LIN {X 0,Y 573.247,Z 310.075,A -85,B 0,C 180,E1 -2008.028,E2 -2008.028} C_VEL
LIN {X 0,Y 573.239,Z 310.078,A -85,B 0,C 180,E1 -2010.176,E2 -2010.176} C_VEL
LIN {X 0,Y 573.253,Z 310.082,A -85,B 0,C 180,E1 -2012.645,E2 -2012.645} C_VEL
LIN {X 0,Y 573.206,Z 310.08,A -85,B 0,C 180,E1 -2015.187,E2 -2015.187} C_VEL
LIN {X 0,Y 573.233,Z 310.076,A -85,B 0,C 180,E1 -2017.807,E2 -2017.807} C_VEL
LIN {X 0,Y 573.244,Z 310.084,A -85,B 0,C 180,E1 -2020.525,E2 -2020.525} C_VEL
LIN {X 0,Y 573.239,Z 310.074,A -85,B 0,C 180,E1 -2023.359,E2 -2023.359} C_VEL
LIN {X 0,Y 573.237,Z 310.083,A -85,B 0,C 180,E1 -2026.331,E2 -2026.331} C_VEL
LIN {X 0,Y 573.228,Z 310.084,A -85,B 0,C 180,E1 -2028.543,E2 -2028.543} C_VEL
LIN {X 0,Y 573.246,Z 310.073,A -85,B 0,C 180,E1 -2031.299,E2 -2031.299} C_VEL
LIN {X 0,Y 573.241,Z 310.079,A -85,B 0,C 180,E1 -2034.014,E2 -2034.014} C_VEL
LIN {X 0,Y 573.284,Z 310.076,A -85,B 0,C 180,E1 -2036.519,E2 -2036.519} C_VEL
LIN {X 0,Y 573.236,Z 310.075,A -85,B 0,C 180,E1 -2039.116,E2 -2039.116} C_VEL
LIN {X 0,Y 573.25,Z 310.078,A -85,B 0,C 180,E1 -2041.971,E2 -2041.971} C_VEL
LIN {X 0,Y 573.255,Z 310.077,A -85,B 0,C 180,E1 -2044.59,E2 -2044.59} C_VEL
LIN {X 0,Y 573.234,Z 310.077,A -85,B 0,C 180,E1 -2047.662,E2 -2047.662} C_VEL
LIN {X 0,Y 573.276,Z 310.072,A -85,B 0,C 180,E1 -2050.728,E2 -2050.728} C_VEL
LIN {X 0,Y 573.247,Z 310.076,A -85,B 0,C 180,E1 -2053.622,E2 -2053.622} C_VEL
LIN {X 0,Y 573.272,Z 310.075,A -85,B 0,C 180,E1 -2055.807,E2 -2055.807} C_VEL
LIN {X 0,Y 573.26,Z 310.073,A -85,B 0,C 180,E1 -2058.745,E2 -2058.745} C_VEL
LIN {X 0,Y 573.282,Z 310.071,A -85,B 0,C 180,E1 -2061.541,E2 -2061.541} C_VEL
LIN {X 0,Y 573.29,Z 310.073,A -85,B 0,C 180,E1 -2064.372,E2 -2064.372} C_VEL
LIN {X 0,Y 573.313,Z 310.073,A -85,B 0,C 180,E1 -2067.893,E2 -2067.893} C_VEL
LIN {X 0,Y 573.33,Z 310.064,A -85,B 0,C 180,E1 -2070.702,E2 -2070.702} C_VEL
LIN {X 0,Y 573.302,Z 310.067,A -85,B 0,C 180,E1 -2072.811,E2 -2072.811} C_VEL
LIN {X 0,Y 573.29,Z 310.073,A -85,B 0,C 180,E1 -2075.628,E2 -2075.628} C_VEL
LIN {X 0,Y 573.282,Z 310.071,A -85,B 0,C 180,E1 -2078.46,E2 -2078.46} C_VEL
LIN {X 0,Y 573.27,Z 310.072,A -85,B 0,C 180,E1 -2081.312,E2 -2081.312} C_VEL
LIN {X 0,Y 573.28,Z 310.071,A -85,B 0,C 180,E1 -2084.425,E2 -2084.425} C_VEL
LIN {X 0,Y 573.258,Z 310.073,A -85,B 0,C 180,E1 -2087.112,E2 -2087.112} C_VEL
LIN {X 0,Y 573.25,Z 310.079,A -85,B 0,C 180,E1 -2090.077,E2 -2090.077} C_VEL
LIN {X 0,Y 573.233,Z 310.076,A -85,B 0,C 180,E1 -2093.1,E2 -2093.1} C_VEL
LIN {X 0,Y 573.255,Z 310.077,A -85,B 0,C 180,E1 -2095.41,E2 -2095.41} C_VEL
LIN {X 0,Y 573.252,Z 310.078,A -85,B 0,C 180,E1 -2098.03,E2 -2098.03} C_VEL
LIN {X 0,Y 573.237,Z 310.075,A -85,B 0,C 180,E1 -2100.884,E2 -2100.884} C_VEL
LIN {X 0,Y 573.262,Z 310.079,A -85,B 0,C 180,E1 -2103.524,E2 -2103.524} C_VEL
LIN {X 0,Y 573.241,Z 310.078,A -85,B 0,C 180,E1 -2106.05,E2 -2106.05} C_VEL
LIN {X 0,Y 573.248,Z 310.073,A -85,B 0,C 180,E1 -2108.702,E2 -2108.702} C_VEL
LIN {X 0,Y 573.229,Z 310.085,A -85,B 0,C 180,E1 -2111.593,E2 -2111.593} C_VEL
LIN {X 0,Y 573.225,Z 310.077,A -85,B 0,C 180,E1 -2114.335,E2 -2114.335} C_VEL
LIN {X 0,Y 573.242,Z 310.081,A -85,B 0,C 180,E1 -2117.359,E2 -2117.359} C_VEL
LIN {X 0,Y 573.24,Z 310.075,A -85,B 0,C 180,E1 -2120.393,E2 -2120.393} C_VEL
LIN {X 0,Y 573.253,Z 310.076,A -85,B 0,C 180,E1 -2123.078,E2 -2123.078} C_VEL
LIN {X 0,Y 573.263,Z 310.078,A -85,B 0,C 180,E1 -2125.671,E2 -2125.671} C_VEL
LIN {X 0,Y 573.241,Z 310.075,A -85,B 0,C 180,E1 -2128.185,E2 -2128.185} C_VEL
LIN {X 0,Y 573.262,Z 310.072,A -85,B 0,C 180,E1 -2130.634,E2 -2130.634} C_VEL
LIN {X 0,Y 573.238,Z 310.083,A -85,B 0,C 180,E1 -2133.509,E2 -2133.509} C_VEL
LIN {X 0,Y 573.225,Z 310.077,A -85,B 0,C 180,E1 -2136.135,E2 -2136.135} C_VEL
LIN {X 0,Y 573.249,Z 310.075,A -85,B 0,C 180,E1 -2138.421,E2 -2138.421} C_VEL
LIN {X 0,Y 573.964,Z 312.69,A -85,B 0,C 180,E1 -2138.478,E2 -2138.478} C_VEL
LIN {X 0,Y 573.861,Z 400.24,A -85,B 0,C 180,E1 -2139.595,E2 -2139.595} C_VEL
LIN {X 0,Y 573.825,Z 411.853,A -85,B 0,C 180,E1 -2139.851,E2 -2139.851} C_VEL
LIN {X 0,Y 573.712,Z 424.112,A -85,B 0,C 180,E1 -2140.248,E2 -2140.248} C_VEL
LIN {X 0,Y 573.584,Z 437.638,A -85,B 0,C 180,E1 -2140.867,E2 -2140.867} C_VEL
LIN {X 0,Y 573.443,Z 448.401,A -85,B 0,C 180,E1 -2141.512,E2 -2141.512} C_VEL
LIN {X 0,Y 573.364,Z 457.219,A -85,B 0,C 180,E1 -2142.156,E2 -2142.156} C_VEL
LIN {X 0,Y 573.312,Z 465.622,A -85,B 0,C 180,E1 -2142.89,E2 -2142.89} C_VEL
LIN {X 0,Y 573.205,Z 472.699,A -85,B 0,C 180,E1 -2143.621,E2 -2143.621} C_VEL
LIN {X 0,Y 573.128,Z 480.104,A -85,B 0,C 180,E1 -2144.532,E2 -2144.532} C_VEL
LIN {X 0,Y 573.081,Z 486.335,A -85,B 0,C 180,E1 -2145.457,E2 -2145.457} C_VEL
LIN {X 0,Y 573.039,Z 492.198,A -85,B 0,C 180,E1 -2146.525,E2 -2146.525} C_VEL
LIN {X 0,Y 573.011,Z 496.871,A -85,B 0,C 180,E1 -2147.606,E2 -2147.606} C_VEL
LIN {X 0,Y 572.987,Z 500.957,A -85,B 0,C 180,E1 -2148.888,E2 -2148.888} C_VEL
LIN {X 0,Y 572.974,Z 503.485,A -85,B 0,C 180,E1 -2150.112,E2 -2150.112} C_VEL
LIN {X 0,Y 572.927,Z 504.386,A -85,B 0,C 180,E1 -2150.824,E2 -2150.824} C_VEL
LIN {X 0,Y 572.978,Z 504.962,A -85,B 0,C 180,E1 -2152.246,E2 -2152.246} C_VEL
LIN {X 0,Y 573.012,Z 504.176,A -85,B 0,C 180,E1 -2153.451,E2 -2153.451} C_VEL
LIN {X 0,Y 573,Z 502.806,A -85,B 0,C 180,E1 -2154.369,E2 -2154.369} C_VEL
LIN {X 0,Y 573.004,Z 500.334,A -85,B 0,C 180,E1 -2155.428,E2 -2155.428} C_VEL
LIN {X 0,Y 573.054,Z 496.866,A -85,B 0,C 180,E1 -2156.485,E2 -2156.485} C_VEL
LIN {X 0,Y 573.033,Z 492.323,A -85,B 0,C 180,E1 -2157.54,E2 -2157.54} C_VEL
LIN {X 0,Y 573.037,Z 486.574,A -85,B 0,C 180,E1 -2158.595,E2 -2158.595} C_VEL
LIN {X 0,Y 573.133,Z 480.729,A -85,B 0,C 180,E1 -2159.473,E2 -2159.473} C_VEL
LIN {X 0,Y 573.178,Z 473.733,A -85,B 0,C 180,E1 -2160.352,E2 -2160.352} C_VEL
LIN {X 0,Y 573.283,Z 465.315,A -85,B 0,C 180,E1 -2161.23,E2 -2161.23} C_VEL
LIN {X 0,Y 573.381,Z 456.163,A -85,B 0,C 180,E1 -2162.02,E2 -2162.02} C_VEL
LIN {X 0,Y 573.481,Z 444.879,A -85,B 0,C 180,E1 -2162.81,E2 -2162.81} C_VEL
LIN {X 0,Y 573.648,Z 433.661,A -85,B 0,C 180,E1 -2163.424,E2 -2163.424} C_VEL
LIN {X 0,Y 573.725,Z 422.252,A -85,B 0,C 180,E1 -2163.907,E2 -2163.907} C_VEL
LIN {X 0,Y 573.768,Z 411.124,A -85,B 0,C 180,E1 -2164.259,E2 -2164.259} C_VEL
LIN {X 0,Y 573.82,Z 399.944,A -85,B 0,C 180,E1 -2164.5,E2 -2164.5} C_VEL
LIN {X 0,Y 573.937,Z 312.624,A -85,B 0,C 180,E1 -2165.614,E2 -2165.614} C_VEL
LIN {X 0,Y 573.248,Z 310.076,A -85,B 0,C 180,E1 -2165.673,E2 -2165.673} C_VEL
LIN {X 0,Y 573.237,Z 310.083,A -85,B 0,C 180,E1 -2168.461,E2 -2168.461} C_VEL
LIN {X 0,Y 573.238,Z 310.076,A -85,B 0,C 180,E1 -2171.313,E2 -2171.313} C_VEL
LIN {X 0,Y 573.262,Z 310.081,A -85,B 0,C 180,E1 -2174.414,E2 -2174.414} C_VEL
LIN {X 0,Y 573.221,Z 310.079,A -85,B 0,C 180,E1 -2177.113,E2 -2177.113} C_VEL
LIN {X 0,Y 573.193,Z 310.086,A -85,B 0,C 180,E1 -2180.079,E2 -2180.079} C_VEL
LIN {X 0,Y 573.223,Z 310.077,A -85,B 0,C 180,E1 -2183.1,E2 -2183.1} C_VEL
LIN {X 0,Y 573.203,Z 310.08,A -85,B 0,C 180,E1 -2185.413,E2 -2185.413} C_VEL
LIN {X 0,Y 573.195,Z 310.087,A -85,B 0,C 180,E1 -2188.017,E2 -2188.017} C_VEL
LIN {X 0,Y 573.216,Z 310.078,A -85,B 0,C 180,E1 -2190.879,E2 -2190.879} C_VEL
LIN {X 0,Y 573.247,Z 310.075,A -85,B 0,C 180,E1 -2193.521,E2 -2193.521} C_VEL
LIN {X 0,Y 573.188,Z 310.09,A -85,B 0,C 180,E1 -2196.054,E2 -2196.054} C_VEL
LIN {X 0,Y 573.234,Z 310.075,A -85,B 0,C 180,E1 -2198.703,E2 -2198.703} C_VEL
LIN {X 0,Y 573.207,Z 310.081,A -85,B 0,C 180,E1 -2201.459,E2 -2201.459} C_VEL
LIN {X 0,Y 573.221,Z 310.08,A -85,B 0,C 180,E1 -2204.335,E2 -2204.335} C_VEL
LIN {X 0,Y 573.233,Z 310.079,A -85,B 0,C 180,E1 -2207.36,E2 -2207.36} C_VEL
LIN {X 0,Y 573.239,Z 310.076,A -85,B 0,C 180,E1 -2210.392,E2 -2210.392} C_VEL
LIN {X 0,Y 573.229,Z 310.078,A -85,B 0,C 180,E1 -2213.075,E2 -2213.075} C_VEL
LIN {X 0,Y 573.263,Z 310.081,A -85,B 0,C 180,E1 -2215.671,E2 -2215.671} C_VEL
LIN {X 0,Y 573.243,Z 310.076,A -85,B 0,C 180,E1 -2218.184,E2 -2218.184} C_VEL
LIN {X 0,Y 573.265,Z 310.073,A -85,B 0,C 180,E1 -2220.634,E2 -2220.634} C_VEL
LIN {X 0,Y 573.265,Z 310.236,A -85,B 0,C 180,E1 -2223.37,E2 -2223.37} C_VEL
LIN {X 0,Y 574.477,Z 315.769,A -85,B 0,C 180,E1 -2224.064,E2 -2224.064} C_VEL
LIN {X 0,Y 574.492,Z 335.278,A -85,B 0,C 180,E1 -2226.319,E2 -2226.319} C_VEL
LIN {X 0,Y 574.163,Z 360.207,A -85,B 0,C 180,E1 -2229.208,E2 -2229.208} C_VEL
LIN {X 0,Y 573.87,Z 385.978,A -85,B 0,C 180,E1 -2232.171,E2 -2232.171} C_VEL
LIN {X 0,Y 573.588,Z 411.75,A -85,B 0,C 180,E1 -2235.089,E2 -2235.089} C_VEL
LIN {X 0,Y 573.505,Z 421.336,A -85,B 0,C 180,E1 -2236.152,E2 -2236.152} C_VEL
LIN {X 0,Y 574.07,Z 426.702,A -85,B 0,C 180,E1 -2236.234,E2 -2236.234} C_VEL
LIN {X 0,Y 573.844,Z 530.936,A -85,B 0,C 180,E1 -2237.556,E2 -2237.556} C_VEL
LIN {X 0,Y 573.767,Z 544.212,A -85,B 0,C 180,E1 -2237.869,E2 -2237.869} C_VEL
LIN {X 0,Y 573.671,Z 557.147,A -85,B 0,C 180,E1 -2238.324,E2 -2238.324} C_VEL
LIN {X 0,Y 573.58,Z 568.667,A -85,B 0,C 180,E1 -2238.875,E2 -2238.875} C_VEL
LIN {X 0,Y 573.435,Z 580.199,A -85,B 0,C 180,E1 -2239.585,E2 -2239.585} C_VEL
LIN {X 0,Y 573.327,Z 590.598,A -85,B 0,C 180,E1 -2240.385,E2 -2240.385} C_VEL
LIN {X 0,Y 573.241,Z 599.111,A -85,B 0,C 180,E1 -2241.184,E2 -2241.184} C_VEL
LIN {X 0,Y 573.161,Z 606.959,A -85,B 0,C 180,E1 -2242.071,E2 -2242.071} C_VEL
LIN {X 0,Y 573.073,Z 614.954,A -85,B 0,C 180,E1 -2243.185,E2 -2243.185} C_VEL
LIN {X 0,Y 573.07,Z 621.679,A -85,B 0,C 180,E1 -2244.369,E2 -2244.369} C_VEL
LIN {X 0,Y 573.029,Z 626.371,A -85,B 0,C 180,E1 -2245.427,E2 -2245.427} C_VEL
LIN {X 0,Y 573.022,Z 629.957,A -85,B 0,C 180,E1 -2246.484,E2 -2246.484} C_VEL
LIN {X 0,Y 572.959,Z 631.808,A -85,B 0,C 180,E1 -2247.188,E2 -2247.188} C_VEL
LIN {X 0,Y 572.938,Z 633.198,A -85,B 0,C 180,E1 -2247.891,E2 -2247.891} C_VEL
LIN {X 0,Y 572.941,Z 634.785,A -85,B 0,C 180,E1 -2249.297,E2 -2249.297} C_VEL
LIN {X 0,Y 572.938,Z 635,A -85,B 0,C 180,E1 -2250,E2 -2250} C_VEL
LIN {X 0,Y 572.946,Z 634.186,A -85,B 0,C 180,E1 -2251.406,E2 -2251.406} C_VEL
LIN {X 0,Y 572.938,Z 633.2,A -85,B 0,C 180,E1 -2252.109,E2 -2252.109} C_VEL
LIN {X 0,Y 572.959,Z 631.81,A -85,B 0,C 180,E1 -2252.812,E2 -2252.812} C_VEL
LIN {X 0,Y 573.014,Z 628.896,A -85,B 0,C 180,E1 -2253.868,E2 -2253.868} C_VEL
LIN {X 0,Y 572.963,Z 624.949,A -85,B 0,C 180,E1 -2254.926,E2 -2254.926} C_VEL
LIN {X 0,Y 573.064,Z 618.877,A -85,B 0,C 180,E1 -2256.16,E2 -2256.16} C_VEL
LIN {X 0,Y 573.119,Z 612.238,A -85,B 0,C 180,E1 -2257.221,E2 -2257.221} C_VEL
LIN {X 0,Y 573.201,Z 603.991,A -85,B 0,C 180,E1 -2258.283,E2 -2258.283} C_VEL
LIN {X 0,Y 573.286,Z 595.539,A -85,B 0,C 180,E1 -2259.17,E2 -2259.17} C_VEL
LIN {X 0,Y 573.423,Z 585.099,A -85,B 0,C 180,E1 -2260.058,E2 -2260.058} C_VEL
LIN {X 0,Y 573.528,Z 573.355,A -85,B 0,C 180,E1 -2260.858,E2 -2260.858} C_VEL
LIN {X 0,Y 573.653,Z 562.283,A -85,B 0,C 180,E1 -2261.447,E2 -2261.447} C_VEL
LIN {X 0,Y 573.746,Z 549.173,A -85,B 0,C 180,E1 -2261.974,E2 -2261.974} C_VEL
LIN {X 0,Y 573.877,Z 536.52,A -85,B 0,C 180,E1 -2262.33,E2 -2262.33} C_VEL
LIN {X 0,Y 573.907,Z 523.312,A -85,B 0,C 180,E1 -2262.554,E2 -2262.554} C_VEL
LIN {X 0,Y 574.014,Z 424.933,A -85,B 0,C 180,E1 -2263.79,E2 -2263.79} C_VEL
LIN {X 0,Y 573.508,Z 421.014,A -85,B 0,C 180,E1 -2263.87,E2 -2263.87} C_VEL
LIN {X 0,Y 573.757,Z 394.034,A -85,B 0,C 180,E1 -2266.913,E2 -2266.913} C_VEL
LIN {X 0,Y 574.033,Z 369.677,A -85,B 0,C 180,E1 -2269.698,E2 -2269.698} C_VEL
LIN {X 0,Y 574.395,Z 344.101,A -85,B 0,C 180,E1 -2272.67,E2 -2272.67} C_VEL
LIN {X 0,Y 574.453,Z 320.232,A -85,B 0,C 180,E1 -2275.353,E2 -2275.353} C_VEL
LIN {X 0,Y 574.306,Z 315.033,A -85,B 0,C 180,E1 -2275.944,E2 -2275.944} C_VEL
LIN {X 0,Y 573.235,Z 310.085,A -85,B 0,C 180,E1 -2276.562,E2 -2276.562} C_VEL
LIN {X 0,Y 573.247,Z 310.075,A -85,B 0,C 180,E1 -2279.488,E2 -2279.488} C_VEL
LIN {X 0,Y 573.255,Z 310.08,A -85,B 0,C 180,E1 -2282.645,E2 -2282.645} C_VEL
LIN {X 0,Y 573.207,Z 310.08,A -85,B 0,C 180,E1 -2285.188,E2 -2285.188} C_VEL
LIN {X 0,Y 573.232,Z 310.078,A -85,B 0,C 180,E1 -2287.808,E2 -2287.808} C_VEL
LIN {X 0,Y 573.248,Z 310.08,A -85,B 0,C 180,E1 -2290.525,E2 -2290.525} C_VEL
LIN {X 0,Y 573.203,Z 310.08,A -85,B 0,C 180,E1 -2293.363,E2 -2293.363} C_VEL
LIN {X 0,Y 573.208,Z 310.085,A -85,B 0,C 180,E1 -2296.335,E2 -2296.335} C_VEL
LIN {X 0,Y 573.206,Z 310.082,A -85,B 0,C 180,E1 -2298.54,E2 -2298.54} C_VEL
LIN {X 0,Y 573.232,Z 310.076,A -85,B 0,C 180,E1 -2301.297,E2 -2301.297} C_VEL
LIN {X 0,Y 573.186,Z 310.09,A -85,B 0,C 180,E1 -2304.023,E2 -2304.023} C_VEL
LIN {X 0,Y 573.224,Z 310.078,A -85,B 0,C 180,E1 -2306.514,E2 -2306.514} C_VEL
LIN {X 0,Y 573.214,Z 310.079,A -85,B 0,C 180,E1 -2309.121,E2 -2309.121} C_VEL
LIN {X 0,Y 573.194,Z 310.087,A -85,B 0,C 180,E1 -2311.983,E2 -2311.983} C_VEL
LIN {X 0,Y 573.201,Z 310.08,A -85,B 0,C 180,E1 -2314.587,E2 -2314.587} C_VEL
LIN {X 0,Y 573.221,Z 310.078,A -85,B 0,C 180,E1 -2316.9,E2 -2316.9} C_VEL
LIN {X 0,Y 573.195,Z 310.085,A -85,B 0,C 180,E1 -2319.921,E2 -2319.921} C_VEL
LIN {X 0,Y 573.216,Z 310.081,A -85,B 0,C 180,E1 -2323.006,E2 -2323.006} C_VEL
LIN {X 0,Y 573.24,Z 310.081,A -85,B 0,C 180,E1 -2325.806,E2 -2325.806} C_VEL
LIN {X 0,Y 573.243,Z 310.142,A -85,B 0,C 180,E1 -2328.428,E2 -2328.428} C_VEL
LIN {X 0,Y 574.02,Z 313.52,A -85,B 0,C 180,E1 -2328.489,E2 -2328.489} C_VEL
LIN {X 0,Y 573.828,Z 401.604,A -85,B 0,C 180,E1 -2329.614,E2 -2329.614} C_VEL
LIN {X 0,Y 573.734,Z 414.619,A -85,B 0,C 180,E1 -2329.925,E2 -2329.925} C_VEL
LIN {X 0,Y 573.665,Z 427.636,A -85,B 0,C 180,E1 -2330.391,E2 -2330.391} C_VEL
LIN {X 0,Y 573.601,Z 438.633,A -85,B 0,C 180,E1 -2330.923,E2 -2330.923} C_VEL
LIN {X 0,Y 573.464,Z 448.855,A -85,B 0,C 180,E1 -2331.543,E2 -2331.543} C_VEL
LIN {X 0,Y 573.347,Z 458.384,A -85,B 0,C 180,E1 -2332.251,E2 -2332.251} C_VEL
LIN {X 0,Y 573.248,Z 467.879,A -85,B 0,C 180,E1 -2333.108,E2 -2333.108} C_VEL
LIN {X 0,Y 573.162,Z 476.135,A -85,B 0,C 180,E1 -2334.017,E2 -2334.017} C_VEL
LIN {X 0,Y 573.152,Z 483.959,A -85,B 0,C 180,E1 -2335.076,E2 -2335.076} C_VEL
LIN {X 0,Y 573.077,Z 490.21,A -85,B 0,C 180,E1 -2336.132,E2 -2336.132} C_VEL
LIN {X 0,Y 572.982,Z 495.189,A -85,B 0,C 180,E1 -2337.187,E2 -2337.187} C_VEL
LIN {X 0,Y 572.995,Z 499.056,A -85,B 0,C 180,E1 -2338.243,E2 -2338.243} C_VEL
LIN {X 0,Y 572.943,Z 501.908,A -85,B 0,C 180,E1 -2339.297,E2 -2339.297} C_VEL
LIN {X 0,Y 572.939,Z 503.308,A -85,B 0,C 180,E1 -2340,E2 -2340} C_VEL
LIN {X 0,Y 572.942,Z 504.25,A -85,B 0,C 180,E1 -2340.703,E2 -2340.703} C_VEL
LIN {X 0,Y 572.936,Z 504.992,A -85,B 0,C 180,E1 -2342.109,E2 -2342.109} C_VEL
LIN {X 0,Y 573.006,Z 504.091,A -85,B 0,C 180,E1 -2343.516,E2 -2343.516} C_VEL
LIN {X 0,Y 573.009,Z 503.098,A -85,B 0,C 180,E1 -2344.22,E2 -2344.22} C_VEL
LIN {X 0,Y 572.945,Z 501.621,A -85,B 0,C 180,E1 -2344.925,E2 -2344.925} C_VEL
LIN {X 0,Y 573.011,Z 498.638,A -85,B 0,C 180,E1 -2345.984,E2 -2345.984} C_VEL
LIN {X 0,Y 573.049,Z 494.615,A -85,B 0,C 180,E1 -2347.044,E2 -2347.044} C_VEL
LIN {X 0,Y 573.084,Z 488.434,A -85,B 0,C 180,E1 -2348.285,E2 -2348.285} C_VEL
LIN {X 0,Y 573.139,Z 481.634,A -85,B 0,C 180,E1 -2349.35,E2 -2349.35} C_VEL
LIN {X 0,Y 573.195,Z 474.703,A -85,B 0,C 180,E1 -2350.24,E2 -2350.24} C_VEL
LIN {X 0,Y 573.257,Z 466.63,A -85,B 0,C 180,E1 -2351.103,E2 -2351.103} C_VEL
LIN {X 0,Y 573.368,Z 458.285,A -85,B 0,C 180,E1 -2351.847,E2 -2351.847} C_VEL
LIN {X 0,Y 573.456,Z 448.609,A -85,B 0,C 180,E1 -2352.564,E2 -2352.564} C_VEL
LIN {X 0,Y 573.577,Z 438.197,A -85,B 0,C 180,E1 -2353.191,E2 -2353.191} C_VEL
LIN {X 0,Y 573.722,Z 424.679,A -85,B 0,C 180,E1 -2353.82,E2 -2353.82} C_VEL
LIN {X 0,Y 573.812,Z 412.467,A -85,B 0,C 180,E1 -2354.223,E2 -2354.223} C_VEL
LIN {X 0,Y 573.861,Z 400.594,A -85,B 0,C 180,E1 -2354.494,E2 -2354.494} C_VEL
LIN {X 0,Y 573.988,Z 345.614,A -85,B 0,C 180,E1 -2355.197,E2 -2355.197} C_VEL
LIN {X 0,Y 573.33,Z 339.807,A -85,B 0,C 180,E1 -2355.286,E2 -2355.286} C_VEL
LIN {X 0,Y 567.786,Z 321.122,A -85,B 0,C 180,E1 -2355.655,E2 -2355.655} C_VEL
LIN {X 0,Y 567.193,Z 315.315,A -85,B 0,C 180,E1 -2355.744,E2 -2355.744} C_VEL
LIN {X 0,Y 566.504,Z 312.222,A -85,B 0,C 180,E1 -2355.801,E2 -2355.801} C_VEL
LIN {X 0,Y 566.215,Z 310.952,A -85,B 0,C 180,E1 -2355.847,E2 -2355.847} C_VEL
LIN {X 0,Y 566.194,Z 310.955,A -85,B 0,C 180,E1 -2358.078,E2 -2358.078} C_VEL
LIN {X 0,Y 566.208,Z 310.955,A -85,B 0,C 180,E1 -2360.337,E2 -2360.337} C_VEL
LIN {X 0,Y 566.169,Z 310.957,A -85,B 0,C 180,E1 -2363.28,E2 -2363.28} C_VEL
LIN {X 0,Y 566.21,Z 310.95,A -85,B 0,C 180,E1 -2365.749,E2 -2365.749} C_VEL
LIN {X 0,Y 566.204,Z 310.954,A -85,B 0,C 180,E1 -2368.202,E2 -2368.202} C_VEL
LIN {X 0,Y 566.188,Z 310.955,A -85,B 0,C 180,E1 -2371.075,E2 -2371.075} C_VEL
LIN {X 0,Y 566.197,Z 310.952,A -85,B 0,C 180,E1 -2373.731,E2 -2373.731} C_VEL
LIN {X 0,Y 566.199,Z 310.961,A -85,B 0,C 180,E1 -2376.569,E2 -2376.569} C_VEL
LIN {X 0,Y 566.214,Z 310.95,A -85,B 0,C 180,E1 -2379.685,E2 -2379.685} C_VEL
LIN {X 0,Y 566.202,Z 310.954,A -85,B 0,C 180,E1 -2382.917,E2 -2382.917} C_VEL
LIN {X 0,Y 566.193,Z 310.956,A -85,B 0,C 180,E1 -2386.049,E2 -2386.049} C_VEL
LIN {X 0,Y 566.202,Z 310.951,A -85,B 0,C 180,E1 -2389.214,E2 -2389.214} C_VEL
LIN {X 0,Y 566.187,Z 310.954,A -85,B 0,C 180,E1 -2391.637,E2 -2391.637} C_VEL
LIN {X 0,Y 566.197,Z 310.96,A -85,B 0,C 180,E1 -2394.31,E2 -2394.31} C_VEL
LIN {X 0,Y 566.227,Z 310.95,A -85,B 0,C 180,E1 -2396.898,E2 -2396.898} C_VEL
LIN {X 0,Y 566.186,Z 310.953,A -85,B 0,C 180,E1 -2399.407,E2 -2399.407} C_VEL
LIN {X 0,Y 566.209,Z 310.954,A -85,B 0,C 180,E1 -2401.857,E2 -2401.857} C_VEL
LIN {X 0,Y 566.214,Z 310.959,A -85,B 0,C 180,E1 -2404.251,E2 -2404.251} C_VEL
LIN {X 0,Y 566.189,Z 310.956,A -85,B 0,C 180,E1 -2406.714,E2 -2406.714} C_VEL
LIN {X 0,Y 566.211,Z 310.952,A -85,B 0,C 180,E1 -2409.663,E2 -2409.663} C_VEL
LIN {X 0,Y 566.201,Z 310.954,A -85,B 0,C 180,E1 -2412.668,E2 -2412.668} C_VEL
LIN {X 0,Y 566.232,Z 310.95,A -85,B 0,C 180,E1 -2415.627,E2 -2415.627} C_VEL
LIN {X 0,Y 566.232,Z 310.949,A -85,B 0,C 180,E1 -2418.675,E2 -2418.675} C_VEL
LIN {X 0,Y 566.226,Z 310.949,A -85,B 0,C 180,E1 -2421.434,E2 -2421.434} C_VEL
LIN {X 0,Y 566.259,Z 310.95,A -85,B 0,C 180,E1 -2424.302,E2 -2424.302} C_VEL
LIN {X 0,Y 566.284,Z 310.948,A -85,B 0,C 180,E1 -2427.866,E2 -2427.866} C_VEL
LIN {X 0,Y 566.3,Z 310.94,A -85,B 0,C 180,E1 -2430.711,E2 -2430.711} C_VEL
LIN {X 0,Y 566.268,Z 310.943,A -85,B 0,C 180,E1 -2432.846,E2 -2432.846} C_VEL
LIN {X 0,Y 566.258,Z 310.95,A -85,B 0,C 180,E1 -2435.698,E2 -2435.698} C_VEL
LIN {X 0,Y 566.226,Z 310.95,A -85,B 0,C 180,E1 -2438.566,E2 -2438.566} C_VEL
LIN {X 0,Y 566.24,Z 310.95,A -85,B 0,C 180,E1 -2441.455,E2 -2441.455} C_VEL
LIN {X 0,Y 566.233,Z 310.949,A -85,B 0,C 180,E1 -2444.507,E2 -2444.507} C_VEL
LIN {X 0,Y 566.202,Z 310.954,A -85,B 0,C 180,E1 -2447.332,E2 -2447.332} C_VEL
LIN {X 0,Y 566.211,Z 310.952,A -85,B 0,C 180,E1 -2450.338,E2 -2450.338} C_VEL
LIN {X 0,Y 566.188,Z 310.957,A -85,B 0,C 180,E1 -2453.404,E2 -2453.404} C_VEL
LIN {X 0,Y 566.215,Z 310.959,A -85,B 0,C 180,E1 -2455.749,E2 -2455.749} C_VEL
LIN {X 0,Y 566.202,Z 310.954,A -85,B 0,C 180,E1 -2458.202,E2 -2458.202} C_VEL
LIN {X 0,Y 566.198,Z 310.953,A -85,B 0,C 180,E1 -2461.078,E2 -2461.078} C_VEL
LIN {X 0,Y 566.212,Z 310.96,A -85,B 0,C 180,E1 -2463.735,E2 -2463.735} C_VEL
LIN {X 0,Y 566.208,Z 310.951,A -85,B 0,C 180,E1 -2466.57,E2 -2466.57} C_VEL
LIN {X 0,Y 566.222,Z 310.958,A -85,B 0,C 180,E1 -2469.687,E2 -2469.687} C_VEL
LIN {X 0,Y 566.201,Z 310.952,A -85,B 0,C 180,E1 -2472.918,E2 -2472.918} C_VEL
LIN {X 0,Y 566.199,Z 310.954,A -85,B 0,C 180,E1 -2476.049,E2 -2476.049} C_VEL
LIN {X 0,Y 566.205,Z 310.956,A -85,B 0,C 180,E1 -2479.215,E2 -2479.215} C_VEL
LIN {X 0,Y 566.186,Z 310.961,A -85,B 0,C 180,E1 -2481.637,E2 -2481.637} C_VEL
LIN {X 0,Y 566.164,Z 310.956,A -85,B 0,C 180,E1 -2484.308,E2 -2484.308} C_VEL
LIN {X 0,Y 566.206,Z 310.953,A -85,B 0,C 180,E1 -2486.897,E2 -2486.897} C_VEL
LIN {X 0,Y 566.177,Z 310.963,A -85,B 0,C 180,E1 -2489.407,E2 -2489.407} C_VEL
LIN {X 0,Y 566.197,Z 310.955,A -85,B 0,C 180,E1 -2491.857,E2 -2491.857} C_VEL
LIN {X 0,Y 566.211,Z 310.95,A -85,B 0,C 180,E1 -2494.251,E2 -2494.251} C_VEL
LIN {X 0,Y 566.171,Z 310.957,A -85,B 0,C 180,E1 -2496.72,E2 -2496.72} C_VEL
LIN {X 0,Y 566.197,Z 310.954,A -85,B 0,C 180,E1 -2498.252,E2 -2498.252} C_VEL
LIN {X 0,Y 567.151,Z 314.922,A -85,B 0,C 180,E1 -2498.34,E2 -2498.34} C_VEL
LIN {X 0,Y 566.961,Z 399.552,A -85,B 0,C 180,E1 -2499.431,E2 -2499.431} C_VEL
LIN {X 0,Y 566.868,Z 410.481,A -85,B 0,C 180,E1 -2499.664,E2 -2499.664} C_VEL
LIN {X 0,Y 566.825,Z 420.39,A -85,B 0,C 180,E1 -2499.97,E2 -2499.97} C_VEL
LIN {X 0,Y 566.689,Z 429.713,A -85,B 0,C 180,E1 -2500.343,E2 -2500.343} C_VEL
LIN {X 0,Y 566.576,Z 439.654,A -85,B 0,C 180,E1 -2500.843,E2 -2500.843} C_VEL
LIN {X 0,Y 566.428,Z 449.574,A -85,B 0,C 180,E1 -2501.462,E2 -2501.462} C_VEL
LIN {X 0,Y 566.335,Z 458.196,A -85,B 0,C 180,E1 -2502.114,E2 -2502.114} C_VEL
LIN {X 0,Y 566.238,Z 466.728,A -85,B 0,C 180,E1 -2502.884,E2 -2502.884} C_VEL
LIN {X 0,Y 566.112,Z 474.987,A -85,B 0,C 180,E1 -2503.78,E2 -2503.78} C_VEL
LIN {X 0,Y 566.045,Z 483.3,A -85,B 0,C 180,E1 -2504.887,E2 -2504.887} C_VEL
LIN {X 0,Y 565.982,Z 489.848,A -85,B 0,C 180,E1 -2505.988,E2 -2505.988} C_VEL
LIN {X 0,Y 565.912,Z 495.009,A -85,B 0,C 180,E1 -2507.083,E2 -2507.083} C_VEL
LIN {X 0,Y 565.906,Z 498.99,A -85,B 0,C 180,E1 -2508.176,E2 -2508.176} C_VEL
LIN {X 0,Y 565.893,Z 501.902,A -85,B 0,C 180,E1 -2509.264,E2 -2509.264} C_VEL
LIN {X 0,Y 565.883,Z 503.33,A -85,B 0,C 180,E1 -2509.987,E2 -2509.987} C_VEL
LIN {X 0,Y 565.829,Z 504.275,A -85,B 0,C 180,E1 -2510.708,E2 -2510.708} C_VEL
LIN {X 0,Y 565.879,Z 504.984,A -85,B 0,C 180,E1 -2512.148,E2 -2512.148} C_VEL
LIN {X 0,Y 565.92,Z 504.17,A -85,B 0,C 180,E1 -2513.466,E2 -2513.466} C_VEL
LIN {X 0,Y 565.905,Z 503.004,A -85,B 0,C 180,E1 -2514.298,E2 -2514.298} C_VEL
LIN {X 0,Y 565.854,Z 501.504,A -85,B 0,C 180,E1 -2515.013,E2 -2515.013} C_VEL
LIN {X 0,Y 565.953,Z 497.254,A -85,B 0,C 180,E1 -2516.441,E2 -2516.441} C_VEL
LIN {X 0,Y 565.957,Z 492.81,A -85,B 0,C 180,E1 -2517.509,E2 -2517.509} C_VEL
LIN {X 0,Y 565.955,Z 487.17,A -85,B 0,C 180,E1 -2518.577,E2 -2518.577} C_VEL
LIN {X 0,Y 566.074,Z 481.443,A -85,B 0,C 180,E1 -2519.467,E2 -2519.467} C_VEL
LIN {X 0,Y 566.115,Z 474.586,A -85,B 0,C 180,E1 -2520.356,E2 -2520.356} C_VEL
LIN {X 0,Y 566.244,Z 466.324,A -85,B 0,C 180,E1 -2521.245,E2 -2521.245} C_VEL
LIN {X 0,Y 566.34,Z 458.444,A -85,B 0,C 180,E1 -2521.956,E2 -2521.956} C_VEL
LIN {X 0,Y 566.45,Z 449.006,A -85,B 0,C 180,E1 -2522.667,E2 -2522.667} C_VEL
LIN {X 0,Y 566.61,Z 438.899,A -85,B 0,C 180,E1 -2523.289,E2 -2523.289} C_VEL
LIN {X 0,Y 566.736,Z 427.103,A -85,B 0,C 180,E1 -2523.867,E2 -2523.867} C_VEL
LIN {X 0,Y 566.813,Z 413.18,A -85,B 0,C 180,E1 -2524.356,E2 -2524.356} C_VEL
LIN {X 0,Y 566.896,Z 401.782,A -85,B 0,C 180,E1 -2524.622,E2 -2524.622} C_VEL
LIN {X 0,Y 566.978,Z 374.049,A -85,B 0,C 180,E1 -2525,E2 -2525} C_VEL
LIN {X 0,Y 567.029,Z 313.898,A -85,B 0,C 180,E1 -2525.766,E2 -2525.766} C_VEL
LIN {X 0,Y 566.216,Z 310.952,A -85,B 0,C 180,E1 -2525.833,E2 -2525.833} C_VEL
LIN {X 0,Y 566.19,Z 310.962,A -85,B 0,C 180,E1 -2528.567,E2 -2528.567} C_VEL
LIN {X 0,Y 566.194,Z 310.954,A -85,B 0,C 180,E1 -2531.456,E2 -2531.456} C_VEL
LIN {X 0,Y 566.218,Z 310.958,A -85,B 0,C 180,E1 -2534.497,E2 -2534.497} C_VEL
LIN {X 0,Y 566.173,Z 310.956,A -85,B 0,C 180,E1 -2537.333,E2 -2537.333} C_VEL
LIN {X 0,Y 566.144,Z 310.968,A -85,B 0,C 180,E1 -2540.34,E2 -2540.34} C_VEL
LIN {X 0,Y 566.17,Z 310.955,A -85,B 0,C 180,E1 -2543.28,E2 -2543.28} C_VEL
LIN {X 0,Y 566.172,Z 310.958,A -85,B 0,C 180,E1 -2545.751,E2 -2545.751} C_VEL
LIN {X 0,Y 566.141,Z 310.968,A -85,B 0,C 180,E1 -2548.189,E2 -2548.189} C_VEL
LIN {X 0,Y 566.18,Z 310.954,A -85,B 0,C 180,E1 -2551.074,E2 -2551.074} C_VEL
LIN {X 0,Y 566.2,Z 310.956,A -85,B 0,C 180,E1 -2553.731,E2 -2553.731} C_VEL
LIN {X 0,Y 566.148,Z 310.959,A -85,B 0,C 180,E1 -2556.574,E2 -2556.574} C_VEL
LIN {X 0,Y 566.21,Z 310.951,A -85,B 0,C 180,E1 -2559.274,E2 -2559.274} C_VEL
LIN {X 0,Y 566.174,Z 310.961,A -85,B 0,C 180,E1 -2562.091,E2 -2562.091} C_VEL
LIN {X 0,Y 566.168,Z 310.956,A -85,B 0,C 180,E1 -2565.037,E2 -2565.037} C_VEL
LIN {X 0,Y 566.183,Z 310.961,A -85,B 0,C 180,E1 -2567.909,E2 -2567.909} C_VEL
LIN {X 0,Y 566.213,Z 310.95,A -85,B 0,C 180,E1 -2570.726,E2 -2570.726} C_VEL
LIN {X 0,Y 566.181,Z 310.96,A -85,B 0,C 180,E1 -2573.428,E2 -2573.428} C_VEL
LIN {X 0,Y 566.201,Z 310.953,A -85,B 0,C 180,E1 -2576.268,E2 -2576.268} C_VEL
LIN {X 0,Y 566.193,Z 310.954,A -85,B 0,C 180,E1 -2578.924,E2 -2578.924} C_VEL
LIN {X 0,Y 566.191,Z 310.96,A -85,B 0,C 180,E1 -2581.856,E2 -2581.856} C_VEL
LIN {X 0,Y 566.19,Z 311.063,A -85,B 0,C 180,E1 -2583.179,E2 -2583.179} C_VEL
LIN {X 0,Y 567.679,Z 318.557,A -85,B 0,C 180,E1 -2584.125,E2 -2584.125} C_VEL
LIN {X 0,Y 567.497,Z 341.924,A -85,B 0,C 180,E1 -2586.846,E2 -2586.846} C_VEL
LIN {X 0,Y 567.243,Z 365.039,A -85,B 0,C 180,E1 -2589.512,E2 -2589.512} C_VEL
LIN {X 0,Y 566.855,Z 392.421,A -85,B 0,C 180,E1 -2592.689,E2 -2592.689} C_VEL
LIN {X 0,Y 566.548,Z 420.609,A -85,B 0,C 180,E1 -2595.91,E2 -2595.91} C_VEL
LIN {X 0,Y 566.613,Z 421.783,A -85,B 0,C 180,E1 -2595.986,E2 -2595.986} C_VEL
LIN {X 0,Y 567.224,Z 428.491,A -85,B 0,C 180,E1 -2596.087,E2 -2596.087} C_VEL
LIN {X 0,Y 566.928,Z 530.935,A -85,B 0,C 180,E1 -2597.402,E2 -2597.402} C_VEL
LIN {X 0,Y 566.853,Z 544.211,A -85,B 0,C 180,E1 -2597.719,E2 -2597.719} C_VEL
LIN {X 0,Y 566.722,Z 557.148,A -85,B 0,C 180,E1 -2598.179,E2 -2598.179} C_VEL
LIN {X 0,Y 566.599,Z 569.363,A -85,B 0,C 180,E1 -2598.776,E2 -2598.776} C_VEL
LIN {X 0,Y 566.424,Z 581.48,A -85,B 0,C 180,E1 -2599.545,E2 -2599.545} C_VEL
LIN {X 0,Y 566.294,Z 591.645,A -85,B 0,C 180,E1 -2600.355,E2 -2600.355} C_VEL
LIN {X 0,Y 566.166,Z 600.785,A -85,B 0,C 180,E1 -2601.253,E2 -2601.253} C_VEL
LIN {X 0,Y 566.081,Z 609.688,A -85,B 0,C 180,E1 -2602.33,E2 -2602.33} C_VEL
LIN {X 0,Y 565.968,Z 616.955,A -85,B 0,C 180,E1 -2603.422,E2 -2603.422} C_VEL
LIN {X 0,Y 566.004,Z 621.679,A -85,B 0,C 180,E1 -2604.299,E2 -2604.299} C_VEL
LIN {X 0,Y 565.933,Z 626.372,A -85,B 0,C 180,E1 -2605.37,E2 -2605.37} C_VEL
LIN {X 0,Y 565.927,Z 629.957,A -85,B 0,C 180,E1 -2606.44,E2 -2606.44} C_VEL
LIN {X 0,Y 565.878,Z 631.808,A -85,B 0,C 180,E1 -2607.152,E2 -2607.152} C_VEL
LIN {X 0,Y 565.846,Z 634.185,A -85,B 0,C 180,E1 -2608.576,E2 -2608.576} C_VEL
LIN {X 0,Y 565.839,Z 635,A -85,B 0,C 180,E1 -2610,E2 -2610} C_VEL
LIN {X 0,Y 565.846,Z 634.186,A -85,B 0,C 180,E1 -2611.423,E2 -2611.423} C_VEL
LIN {X 0,Y 565.878,Z 631.81,A -85,B 0,C 180,E1 -2612.847,E2 -2612.847} C_VEL
LIN {X 0,Y 565.926,Z 628.896,A -85,B 0,C 180,E1 -2613.916,E2 -2613.916} C_VEL
LIN {X 0,Y 565.878,Z 624.949,A -85,B 0,C 180,E1 -2614.987,E2 -2614.987} C_VEL
LIN {X 0,Y 566.002,Z 619.867,A -85,B 0,C 180,E1 -2616.058,E2 -2616.058} C_VEL
LIN {X 0,Y 566.04,Z 613.469,A -85,B 0,C 180,E1 -2617.132,E2 -2617.132} C_VEL
LIN {X 0,Y 566.134,Z 605.479,A -85,B 0,C 180,E1 -2618.208,E2 -2618.208} C_VEL
LIN {X 0,Y 566.228,Z 597.336,A -85,B 0,C 180,E1 -2619.105,E2 -2619.105} C_VEL
LIN {X 0,Y 566.343,Z 587.401,A -85,B 0,C 180,E1 -2620.005,E2 -2620.005} C_VEL
LIN {X 0,Y 566.529,Z 576.291,A -85,B 0,C 180,E1 -2620.807,E2 -2620.807} C_VEL
LIN {X 0,Y 566.613,Z 565.176,A -85,B 0,C 180,E1 -2621.447,E2 -2621.447} C_VEL
LIN {X 0,Y 566.737,Z 552.983,A -85,B 0,C 180,E1 -2621.988,E2 -2621.988} C_VEL
LIN {X 0,Y 566.884,Z 540.177,A -85,B 0,C 180,E1 -2622.394,E2 -2622.394} C_VEL
LIN {X 0,Y 566.974,Z 526.603,A -85,B 0,C 180,E1 -2622.665,E2 -2622.665} C_VEL
LIN {X 0,Y 567.124,Z 425.604,A -85,B 0,C 180,E1 -2623.953,E2 -2623.953} C_VEL
LIN {X 0,Y 566.536,Z 421.014,A -85,B 0,C 180,E1 -2624.045,E2 -2624.045} C_VEL
LIN {X 0,Y 566.837,Z 393.552,A -85,B 0,C 180,E1 -2627.181,E2 -2627.181} C_VEL
LIN {X 0,Y 567.182,Z 368.264,A -85,B 0,C 180,E1 -2630.112,E2 -2630.112} C_VEL
LIN {X 0,Y 567.365,Z 350.067,A -85,B 0,C 180,E1 -2632.198,E2 -2632.198} C_VEL
LIN {X 0,Y 567.508,Z 326.08,A -85,B 0,C 180,E1 -2634.901,E2 -2634.901} C_VEL
LIN {X 0,Y 567.472,Z 317.453,A -85,B 0,C 180,E1 -2635.885,E2 -2635.885} C_VEL
LIN {X 0,Y 566.205,Z 310.96,A -85,B 0,C 180,E1 -2636.693,E2 -2636.693} C_VEL
LIN {X 0,Y 566.203,Z 310.954,A -85,B 0,C 180,E1 -2639.769,E2 -2639.769} C_VEL
LIN {X 0,Y 566.206,Z 310.961,A -85,B 0,C 180,E1 -2642.43,E2 -2642.43} C_VEL
LIN {X 0,Y 566.179,Z 310.956,A -85,B 0,C 180,E1 -2644.989,E2 -2644.989} C_VEL
LIN {X 0,Y 566.194,Z 310.953,A -85,B 0,C 180,E1 -2647.461,E2 -2647.461} C_VEL
LIN {X 0,Y 566.209,Z 310.96,A -85,B 0,C 180,E1 -2650.199,E2 -2650.199} C_VEL
LIN {X 0,Y 566.184,Z 310.954,A -85,B 0,C 180,E1 -2653.056,E2 -2653.056} C_VEL
LIN {X 0,Y 566.16,Z 310.966,A -85,B 0,C 180,E1 -2656.053,E2 -2656.053} C_VEL
LIN {X 0,Y 566.159,Z 310.957,A -85,B 0,C 180,E1 -2658.859,E2 -2658.859} C_VEL
LIN {X 0,Y 566.203,Z 310.953,A -85,B 0,C 180,E1 -2661.443,E2 -2661.443} C_VEL
LIN {X 0,Y 566.14,Z 310.963,A -85,B 0,C 180,E1 -2664.306,E2 -2664.306} C_VEL
LIN {X 0,Y 566.194,Z 310.952,A -85,B 0,C 180,E1 -2666.896,E2 -2666.896} C_VEL
LIN {X 0,Y 566.163,Z 310.96,A -85,B 0,C 180,E1 -2669.406,E2 -2669.406} C_VEL
LIN {X 0,Y 566.141,Z 310.968,A -85,B 0,C 180,E1 -2671.853,E2 -2671.853} C_VEL
LIN {X 0,Y 566.171,Z 310.958,A -85,B 0,C 180,E1 -2674.249,E2 -2674.249} C_VEL
LIN {X 0,Y 566.168,Z 310.956,A -85,B 0,C 180,E1 -2676.72,E2 -2676.72} C_VEL
LIN {X 0,Y 566.144,Z 310.967,A -85,B 0,C 180,E1 -2679.66,E2 -2679.66} C_VEL
LIN {X 0,Y 566.161,Z 310.961,A -85,B 0,C 180,E1 -2681.92,E2 -2681.92} C_VEL
LIN {X 0,Y 566.182,Z 310.957,A -85,B 0,C 180,E1 -2684.89,E2 -2684.89} C_VEL
LIN {X 0,Y 566.179,Z 310.96,A -85,B 0,C 180,E1 -2687.817,E2 -2687.817} C_VEL
LIN {X 0,Y 566.223,Z 310.951,A -85,B 0,C 180,E1 -2688.263,E2 -2688.263} C_VEL
LIN {X 0,Y 567.133,Z 314.807,A -85,B 0,C 180,E1 -2688.338,E2 -2688.338} C_VEL
LIN {X 0,Y 566.919,Z 400.625,A -85,B 0,C 180,E1 -2689.441,E2 -2689.441} C_VEL
LIN {X 0,Y 566.79,Z 413.077,A -85,B 0,C 180,E1 -2689.732,E2 -2689.732} C_VEL
LIN {X 0,Y 566.706,Z 426.14,A -85,B 0,C 180,E1 -2690.182,E2 -2690.182} C_VEL
LIN {X 0,Y 566.631,Z 437.504,A -85,B 0,C 180,E1 -2690.721,E2 -2690.721} C_VEL
LIN {X 0,Y 566.452,Z 447.92,A -85,B 0,C 180,E1 -2691.348,E2 -2691.348} C_VEL
LIN {X 0,Y 566.364,Z 457.598,A -85,B 0,C 180,E1 -2692.065,E2 -2692.065} C_VEL
LIN {X 0,Y 566.281,Z 464.749,A -85,B 0,C 180,E1 -2692.691,E2 -2692.691} C_VEL
LIN {X 0,Y 566.192,Z 473.292,A -85,B 0,C 180,E1 -2693.585,E2 -2693.585} C_VEL
LIN {X 0,Y 566.024,Z 480.389,A -85,B 0,C 180,E1 -2694.478,E2 -2694.478} C_VEL
LIN {X 0,Y 566.033,Z 486.301,A -85,B 0,C 180,E1 -2695.371,E2 -2695.371} C_VEL
LIN {X 0,Y 565.996,Z 492.107,A -85,B 0,C 180,E1 -2696.44,E2 -2696.44} C_VEL
LIN {X 0,Y 565.954,Z 496.695,A -85,B 0,C 180,E1 -2697.509,E2 -2697.509} C_VEL
LIN {X 0,Y 565.863,Z 500.199,A -85,B 0,C 180,E1 -2698.576,E2 -2698.576} C_VEL
LIN {X 0,Y 565.839,Z 503.349,A -85,B 0,C 180,E1 -2700,E2 -2700} C_VEL
LIN {X 0,Y 565.842,Z 504.277,A -85,B 0,C 180,E1 -2700.711,E2 -2700.711} C_VEL
LIN {X 0,Y 565.837,Z 504.986,A -85,B 0,C 180,E1 -2702.135,E2 -2702.135} C_VEL
LIN {X 0,Y 565.873,Z 504.718,A -85,B 0,C 180,E1 -2702.847,E2 -2702.847} C_VEL
LIN {X 0,Y 565.913,Z 503.05,A -85,B 0,C 180,E1 -2704.273,E2 -2704.273} C_VEL
LIN {X 0,Y 565.859,Z 501.557,A -85,B 0,C 180,E1 -2704.987,E2 -2704.987} C_VEL
LIN {X 0,Y 565.918,Z 497.344,A -85,B 0,C 180,E1 -2706.417,E2 -2706.417} C_VEL
LIN {X 0,Y 565.974,Z 492.897,A -85,B 0,C 180,E1 -2707.491,E2 -2707.491} C_VEL
LIN {X 0,Y 566.013,Z 487.216,A -85,B 0,C 180,E1 -2708.569,E2 -2708.569} C_VEL
LIN {X 0,Y 566.064,Z 481.432,A -85,B 0,C 180,E1 -2709.468,E2 -2709.468} C_VEL
LIN {X 0,Y 566.159,Z 474.464,A -85,B 0,C 180,E1 -2710.369,E2 -2710.369} C_VEL
LIN {X 0,Y 566.215,Z 467.148,A -85,B 0,C 180,E1 -2711.165,E2 -2711.165} C_VEL
LIN {X 0,Y 566.334,Z 459.051,A -85,B 0,C 180,E1 -2711.906,E2 -2711.906} C_VEL
LIN {X 0,Y 566.45,Z 449.528,A -85,B 0,C 180,E1 -2712.631,E2 -2712.631} C_VEL
LIN {X 0,Y 566.556,Z 440.905,A -85,B 0,C 180,E1 -2713.175,E2 -2713.175} C_VEL
LIN {X 0,Y 566.686,Z 432.28,A -85,B 0,C 180,E1 -2713.629,E2 -2713.629} C_VEL
LIN {X 0,Y 566.813,Z 422.69,A -85,B 0,C 180,E1 -2714.037,E2 -2714.037} C_VEL
LIN {X 0,Y 566.86,Z 411.658,A -85,B 0,C 180,E1 -2714.395,E2 -2714.395} C_VEL
LIN {X 0,Y 566.942,Z 400.621,A -85,B 0,C 180,E1 -2714.648,E2 -2714.648} C_VEL
LIN {X 0,Y 567.193,Z 315.315,A -85,B 0,C 180,E1 -2715.744,E2 -2715.744} C_VEL
LIN {X 0,Y 566.89,Z 313.363,A -85,B 0,C 180,E1 -2715.851,E2 -2715.851} C_VEL
LIN {X 0,Y 565.95,Z 311.824,A -85,B 0,C 180,E1 -2716.118,E2 -2716.118} C_VEL
LIN {X 0,Y 564.378,Z 311.235,A -85,B 0,C 180,E1 -2716.551,E2 -2716.551} C_VEL
LIN {X 0,Y 560.364,Z 311.748,A -85,B 0,C 180,E1 -2717.845,E2 -2717.845} C_VEL
LIN {X 0,Y 559.224,Z 311.831,A -85,B 0,C 180,E1 -2718.564,E2 -2718.564} C_VEL
LIN {X 0,Y 559.144,Z 311.834,A -85,B 0,C 180,E1 -2718.807,E2 -2718.807} C_VEL
LIN {X 0,Y 559.157,Z 311.829,A -85,B 0,C 180,E1 -2721.549,E2 -2721.549} C_VEL
LIN {X 0,Y 559.155,Z 311.836,A -85,B 0,C 180,E1 -2724.505,E2 -2724.505} C_VEL
LIN {X 0,Y 559.169,Z 311.833,A -85,B 0,C 180,E1 -2726.902,E2 -2726.902} C_VEL
LIN {X 0,Y 559.145,Z 311.831,A -85,B 0,C 180,E1 -2729.856,E2 -2729.856} C_VEL
LIN {X 0,Y 559.153,Z 311.837,A -85,B 0,C 180,E1 -2732.715,E2 -2732.715} C_VEL
LIN {X 0,Y 559.127,Z 311.833,A -85,B 0,C 180,E1 -2735.324,E2 -2735.324} C_VEL
LIN {X 0,Y 559.132,Z 311.834,A -85,B 0,C 180,E1 -2738.017,E2 -2738.017} C_VEL
LIN {X 0,Y 559.155,Z 311.834,A -85,B 0,C 180,E1 -2740.812,E2 -2740.812} C_VEL
LIN {X 0,Y 559.14,Z 311.832,A -85,B 0,C 180,E1 -2743.733,E2 -2743.733} C_VEL
LIN {X 0,Y 559.143,Z 311.835,A -85,B 0,C 180,E1 -2746.803,E2 -2746.803} C_VEL
LIN {X 0,Y 559.154,Z 311.83,A -85,B 0,C 180,E1 -2749.187,E2 -2749.187} C_VEL
LIN {X 0,Y 559.132,Z 311.836,A -85,B 0,C 180,E1 -2751.982,E2 -2751.982} C_VEL
LIN {X 0,Y 559.153,Z 311.833,A -85,B 0,C 180,E1 -2754.783,E2 -2754.783} C_VEL
LIN {X 0,Y 559.172,Z 311.827,A -85,B 0,C 180,E1 -2757.361,E2 -2757.361} C_VEL
LIN {X 0,Y 559.148,Z 311.837,A -85,B 0,C 180,E1 -2760.142,E2 -2760.142} C_VEL
LIN {X 0,Y 559.168,Z 311.828,A -85,B 0,C 180,E1 -2763.098,E2 -2763.098} C_VEL
LIN {X 0,Y 559.155,Z 311.83,A -85,B 0,C 180,E1 -2765.495,E2 -2765.495} C_VEL
LIN {X 0,Y 559.169,Z 311.831,A -85,B 0,C 180,E1 -2768.624,E2 -2768.624} C_VEL
LIN {X 0,Y 559.167,Z 311.828,A -85,B 0,C 180,E1 -2770.926,E2 -2770.926} C_VEL
LIN {X 0,Y 559.164,Z 311.834,A -85,B 0,C 180,E1 -2773.948,E2 -2773.948} C_VEL
LIN {X 0,Y 559.17,Z 311.837,A -85,B 0,C 180,E1 -2776.184,E2 -2776.184} C_VEL
LIN {X 0,Y 559.194,Z 311.824,A -85,B 0,C 180,E1 -2779.134,E2 -2779.134} C_VEL
LIN {X 0,Y 559.202,Z 311.832,A -85,B 0,C 180,E1 -2782.054,E2 -2782.054} C_VEL
LIN {X 0,Y 559.25,Z 311.817,A -85,B 0,C 180,E1 -2784.953,E2 -2784.953} C_VEL
LIN {X 0,Y 559.254,Z 311.823,A -85,B 0,C 180,E1 -2787.84,E2 -2787.84} C_VEL
LIN {X 0,Y 559.27,Z 311.816,A -85,B 0,C 180,E1 -2790.72,E2 -2790.72} C_VEL
LIN {X 0,Y 559.235,Z 311.819,A -85,B 0,C 180,E1 -2792.882,E2 -2792.882} C_VEL
LIN {X 0,Y 559.227,Z 311.827,A -85,B 0,C 180,E1 -2795.77,E2 -2795.77} C_VEL
LIN {X 0,Y 559.185,Z 311.826,A -85,B 0,C 180,E1 -2798.675,E2 -2798.675} C_VEL
LIN {X 0,Y 559.204,Z 311.828,A -85,B 0,C 180,E1 -2801.601,E2 -2801.601} C_VEL
LIN {X 0,Y 559.198,Z 311.825,A -85,B 0,C 180,E1 -2804.596,E2 -2804.596} C_VEL
LIN {X 0,Y 559.161,Z 311.834,A -85,B 0,C 180,E1 -2807.557,E2 -2807.557} C_VEL
LIN {X 0,Y 559.171,Z 311.836,A -85,B 0,C 180,E1 -2809.838,E2 -2809.838} C_VEL
LIN {X 0,Y 559.139,Z 311.835,A -85,B 0,C 180,E1 -2812.153,E2 -2812.153} C_VEL
LIN {X 0,Y 559.178,Z 311.828,A -85,B 0,C 180,E1 -2815.187,E2 -2815.187} C_VEL
LIN {X 0,Y 559.18,Z 311.834,A -85,B 0,C 180,E1 -2817.713,E2 -2817.713} C_VEL
LIN {X 0,Y 559.156,Z 311.832,A -85,B 0,C 180,E1 -2820.183,E2 -2820.183} C_VEL
LIN {X 0,Y 559.175,Z 311.827,A -85,B 0,C 180,E1 -2822.714,E2 -2822.714} C_VEL
LIN {X 0,Y 559.15,Z 311.834,A -85,B 0,C 180,E1 -2825.323,E2 -2825.323} C_VEL
LIN {X 0,Y 559.134,Z 311.836,A -85,B 0,C 180,E1 -2828.018,E2 -2828.018} C_VEL
LIN {X 0,Y 559.155,Z 311.83,A -85,B 0,C 180,E1 -2830.813,E2 -2830.813} C_VEL
LIN {X 0,Y 559.138,Z 311.839,A -85,B 0,C 180,E1 -2833.735,E2 -2833.735} C_VEL
LIN {X 0,Y 559.148,Z 311.831,A -85,B 0,C 180,E1 -2836.804,E2 -2836.804} C_VEL
LIN {X 0,Y 559.156,Z 311.833,A -85,B 0,C 180,E1 -2839.188,E2 -2839.188} C_VEL
LIN {X 0,Y 559.134,Z 311.835,A -85,B 0,C 180,E1 -2841.983,E2 -2841.983} C_VEL
LIN {X 0,Y 559.133,Z 311.833,A -85,B 0,C 180,E1 -2844.788,E2 -2844.788} C_VEL
LIN {X 0,Y 559.156,Z 311.837,A -85,B 0,C 180,E1 -2847.365,E2 -2847.365} C_VEL
LIN {X 0,Y 559.147,Z 311.831,A -85,B 0,C 180,E1 -2850.144,E2 -2850.144} C_VEL
LIN {X 0,Y 559.167,Z 311.833,A -85,B 0,C 180,E1 -2853.098,E2 -2853.098} C_VEL
LIN {X 0,Y 559.158,Z 311.837,A -85,B 0,C 180,E1 -2855.495,E2 -2855.495} C_VEL
LIN {X 0,Y 559.163,Z 311.832,A -85,B 0,C 180,E1 -2858.085,E2 -2858.085} C_VEL
LIN {X 0,Y 560.236,Z 315.429,A -85,B 0,C 180,E1 -2858.174,E2 -2858.174} C_VEL
LIN {X 0,Y 560.031,Z 400.211,A -85,B 0,C 180,E1 -2859.285,E2 -2859.285} C_VEL
LIN {X 0,Y 559.953,Z 410.027,A -85,B 0,C 180,E1 -2859.498,E2 -2859.498} C_VEL
LIN {X 0,Y 559.885,Z 420.053,A -85,B 0,C 180,E1 -2859.807,E2 -2859.807} C_VEL
LIN {X 0,Y 559.721,Z 429.447,A -85,B 0,C 180,E1 -2860.183,E2 -2860.183} C_VEL
LIN {X 0,Y 559.624,Z 438.714,A -85,B 0,C 180,E1 -2860.649,E2 -2860.649} C_VEL
LIN {X 0,Y 559.486,Z 448.045,A -85,B 0,C 180,E1 -2861.223,E2 -2861.223} C_VEL
LIN {X 0,Y 559.336,Z 456.911,A -85,B 0,C 180,E1 -2861.882,E2 -2861.882} C_VEL
LIN {X 0,Y 559.238,Z 465.673,A -85,B 0,C 180,E1 -2862.666,E2 -2862.666} C_VEL
LIN {X 0,Y 559.131,Z 472.48,A -85,B 0,C 180,E1 -2863.384,E2 -2863.384} C_VEL
LIN {X 0,Y 559.013,Z 479.917,A -85,B 0,C 180,E1 -2864.318,E2 -2864.318} C_VEL
LIN {X 0,Y 558.928,Z 486.073,A -85,B 0,C 180,E1 -2865.249,E2 -2865.249} C_VEL
LIN {X 0,Y 558.869,Z 491.158,A -85,B 0,C 180,E1 -2866.177,E2 -2866.177} C_VEL
LIN {X 0,Y 558.829,Z 496.045,A -85,B 0,C 180,E1 -2867.286,E2 -2867.286} C_VEL
LIN {X 0,Y 558.837,Z 499.776,A -85,B 0,C 180,E1 -2868.392,E2 -2868.392} C_VEL
LIN {X 0,Y 558.794,Z 501.677,A -85,B 0,C 180,E1 -2869.126,E2 -2869.126} C_VEL
LIN {X 0,Y 558.779,Z 503.175,A -85,B 0,C 180,E1 -2869.859,E2 -2869.859} C_VEL
LIN {X 0,Y 558.766,Z 504.746,A -85,B 0,C 180,E1 -2871.319,E2 -2871.319} C_VEL
LIN {X 0,Y 558.797,Z 505,A -85,B 0,C 180,E1 -2872.048,E2 -2872.048} C_VEL
LIN {X 0,Y 558.827,Z 504.139,A -85,B 0,C 180,E1 -2873.501,E2 -2873.501} C_VEL
LIN {X 0,Y 558.816,Z 503.183,A -85,B 0,C 180,E1 -2874.226,E2 -2874.226} C_VEL
LIN {X 0,Y 558.828,Z 499.851,A -85,B 0,C 180,E1 -2875.673,E2 -2875.673} C_VEL
LIN {X 0,Y 558.856,Z 496.23,A -85,B 0,C 180,E1 -2876.756,E2 -2876.756} C_VEL
LIN {X 0,Y 558.82,Z 491.53,A -85,B 0,C 180,E1 -2877.838,E2 -2877.838} C_VEL
LIN {X 0,Y 558.946,Z 485.6,A -85,B 0,C 180,E1 -2878.92,E2 -2878.92} C_VEL
LIN {X 0,Y 559.033,Z 478.273,A -85,B 0,C 180,E1 -2880,E2 -2880} C_VEL
LIN {X 0,Y 559.173,Z 469.14,A -85,B 0,C 180,E1 -2881.081,E2 -2881.081} C_VEL
LIN {X 0,Y 559.312,Z 459.642,A -85,B 0,C 180,E1 -2881.981,E2 -2881.981} C_VEL
LIN {X 0,Y 559.438,Z 450.438,A -85,B 0,C 180,E1 -2882.701,E2 -2882.701} C_VEL
LIN {X 0,Y 559.589,Z 442.2,A -85,B 0,C 180,E1 -2883.24,E2 -2883.24} C_VEL
LIN {X 0,Y 559.734,Z 432.153,A -85,B 0,C 180,E1 -2883.78,E2 -2883.78} C_VEL
LIN {X 0,Y 559.827,Z 422.788,A -85,B 0,C 180,E1 -2884.185,E2 -2884.185} C_VEL
LIN {X 0,Y 559.897,Z 411.844,A -85,B 0,C 180,E1 -2884.545,E2 -2884.545} C_VEL
LIN {X 0,Y 559.96,Z 401.046,A -85,B 0,C 180,E1 -2884.793,E2 -2884.793} C_VEL
LIN {X 0,Y 560.146,Z 357.296,A -85,B 0,C 180,E1 -2885.377,E2 -2885.377} C_VEL
LIN {X 0,Y 560.225,Z 315.415,A -85,B 0,C 180,E1 -2885.916,E2 -2885.916} C_VEL
LIN {X 0,Y 559.177,Z 311.83,A -85,B 0,C 180,E1 -2885.997,E2 -2885.997} C_VEL
LIN {X 0,Y 559.156,Z 311.839,A -85,B 0,C 180,E1 -2888.675,E2 -2888.675} C_VEL
LIN {X 0,Y 559.135,Z 311.833,A -85,B 0,C 180,E1 -2891.602,E2 -2891.602} C_VEL
LIN {X 0,Y 559.164,Z 311.837,A -85,B 0,C 180,E1 -2894.579,E2 -2894.579} C_VEL
LIN {X 0,Y 559.121,Z 311.835,A -85,B 0,C 180,E1 -2897.558,E2 -2897.558} C_VEL
LIN {X 0,Y 559.108,Z 311.839,A -85,B 0,C 180,E1 -2899.84,E2 -2899.84} C_VEL
LIN {X 0,Y 559.109,Z 311.843,A -85,B 0,C 180,E1 -2902.154,E2 -2902.154} C_VEL
LIN {X 0,Y 559.102,Z 311.843,A -85,B 0,C 180,E1 -2904.508,E2 -2904.508} C_VEL
LIN {X 0,Y 559.112,Z 311.836,A -85,B 0,C 180,E1 -2906.906,E2 -2906.906} C_VEL
LIN {X 0,Y 559.111,Z 311.839,A -85,B 0,C 180,E1 -2909.85,E2 -2909.85} C_VEL
LIN {X 0,Y 559.152,Z 311.831,A -85,B 0,C 180,E1 -2912.716,E2 -2912.716} C_VEL
LIN {X 0,Y 559.118,Z 311.834,A -85,B 0,C 180,E1 -2915.325,E2 -2915.325} C_VEL
LIN {X 0,Y 559.127,Z 311.841,A -85,B 0,C 180,E1 -2918.018,E2 -2918.018} C_VEL
LIN {X 0,Y 559.13,Z 311.831,A -85,B 0,C 180,E1 -2920.815,E2 -2920.815} C_VEL
LIN {X 0,Y 559.129,Z 311.833,A -85,B 0,C 180,E1 -2923.194,E2 -2923.194} C_VEL
LIN {X 0,Y 559.128,Z 311.841,A -85,B 0,C 180,E1 -2925.764,E2 -2925.764} C_VEL
LIN {X 0,Y 559.129,Z 311.835,A -85,B 0,C 180,E1 -2928.226,E2 -2928.226} C_VEL
LIN {X 0,Y 559.174,Z 311.829,A -85,B 0,C 180,E1 -2931.192,E2 -2931.192} C_VEL
LIN {X 0,Y 559.122,Z 311.841,A -85,B 0,C 180,E1 -2933.787,E2 -2933.787} C_VEL
LIN {X 0,Y 559.152,Z 311.83,A -85,B 0,C 180,E1 -2936.424,E2 -2936.424} C_VEL
LIN {X 0,Y 559.158,Z 311.831,A -85,B 0,C 180,E1 -2938.98,E2 -2938.98} C_VEL
LIN {X 0,Y 559.138,Z 311.841,A -85,B 0,C 180,E1 -2941.625,E2 -2941.625} C_VEL
LIN {X 0,Y 559.164,Z 311.987,A -85,B 0,C 180,E1 -2942.996,E2 -2942.996} C_VEL
LIN {X 0,Y 560.767,Z 319.66,A -85,B 0,C 180,E1 -2943.982,E2 -2943.982} C_VEL
LIN {X 0,Y 560.594,Z 339.697,A -85,B 0,C 180,E1 -2946.348,E2 -2946.348} C_VEL
LIN {X 0,Y 560.316,Z 364.577,A -85,B 0,C 180,E1 -2949.247,E2 -2949.247} C_VEL
LIN {X 0,Y 559.989,Z 389.2,A -85,B 0,C 180,E1 -2952.092,E2 -2952.092} C_VEL
LIN {X 0,Y 559.605,Z 415.004,A -85,B 0,C 180,E1 -2955.084,E2 -2955.084} C_VEL
LIN {X 0,Y 559.566,Z 421.336,A -85,B 0,C 180,E1 -2955.8,E2 -2955.8} C_VEL
LIN {X 0,Y 560.349,Z 428.491,A -85,B 0,C 180,E1 -2955.913,E2 -2955.913} C_VEL
LIN {X 0,Y 560.023,Z 530.935,A -85,B 0,C 180,E1 -2957.244,E2 -2957.244} C_VEL
LIN {X 0,Y 559.92,Z 544.211,A -85,B 0,C 180,E1 -2957.564,E2 -2957.564} C_VEL
LIN {X 0,Y 559.77,Z 557.15,A -85,B 0,C 180,E1 -2958.03,E2 -2958.03} C_VEL
LIN {X 0,Y 559.6,Z 569.461,A -85,B 0,C 180,E1 -2958.64,E2 -2958.64} C_VEL
LIN {X 0,Y 559.433,Z 581.482,A -85,B 0,C 180,E1 -2959.413,E2 -2959.413} C_VEL
LIN {X 0,Y 559.289,Z 591.644,A -85,B 0,C 180,E1 -2960.233,E2 -2960.233} C_VEL
LIN {X 0,Y 559.135,Z 600.784,A -85,B 0,C 180,E1 -2961.142,E2 -2961.142} C_VEL
LIN {X 0,Y 559.01,Z 609.687,A -85,B 0,C 180,E1 -2962.232,E2 -2962.232} C_VEL
LIN {X 0,Y 558.925,Z 615.739,A -85,B 0,C 180,E1 -2963.14,E2 -2963.14} C_VEL
LIN {X 0,Y 558.935,Z 621.679,A -85,B 0,C 180,E1 -2964.227,E2 -2964.227} C_VEL
LIN {X 0,Y 558.827,Z 626.372,A -85,B 0,C 180,E1 -2965.311,E2 -2965.311} C_VEL
LIN {X 0,Y 558.836,Z 629.957,A -85,B 0,C 180,E1 -2966.395,E2 -2966.395} C_VEL
LIN {X 0,Y 558.799,Z 631.807,A -85,B 0,C 180,E1 -2967.116,E2 -2967.116} C_VEL
LIN {X 0,Y 558.745,Z 634.184,A -85,B 0,C 180,E1 -2968.558,E2 -2968.558} C_VEL
LIN {X 0,Y 558.74,Z 635,A -85,B 0,C 180,E1 -2970,E2 -2970} C_VEL
LIN {X 0,Y 558.745,Z 634.185,A -85,B 0,C 180,E1 -2971.441,E2 -2971.441} C_VEL
LIN {X 0,Y 558.799,Z 631.81,A -85,B 0,C 180,E1 -2972.884,E2 -2972.884} C_VEL
LIN {X 0,Y 558.844,Z 628.896,A -85,B 0,C 180,E1 -2973.966,E2 -2973.966} C_VEL
LIN {X 0,Y 558.799,Z 624.949,A -85,B 0,C 180,E1 -2975.051,E2 -2975.051} C_VEL
LIN {X 0,Y 558.921,Z 619.867,A -85,B 0,C 180,E1 -2976.135,E2 -2976.135} C_VEL
LIN {X 0,Y 558.977,Z 613.468,A -85,B 0,C 180,E1 -2977.223,E2 -2977.223} C_VEL
LIN {X 0,Y 559.099,Z 605.478,A -85,B 0,C 180,E1 -2978.312,E2 -2978.312} C_VEL
LIN {X 0,Y 559.184,Z 597.335,A -85,B 0,C 180,E1 -2979.221,E2 -2979.221} C_VEL
LIN {X 0,Y 559.356,Z 587.4,A -85,B 0,C 180,E1 -2980.131,E2 -2980.131} C_VEL
LIN {X 0,Y 559.543,Z 576.4,A -85,B 0,C 180,E1 -2980.937,E2 -2980.937} C_VEL
LIN {X 0,Y 559.672,Z 564.461,A -85,B 0,C 180,E1 -2981.628,E2 -2981.628} C_VEL
LIN {X 0,Y 559.822,Z 551.769,A -85,B 0,C 180,E1 -2982.185,E2 -2982.185} C_VEL
LIN {X 0,Y 560.005,Z 538.347,A -85,B 0,C 180,E1 -2982.595,E2 -2982.595} C_VEL
LIN {X 0,Y 560.057,Z 525.086,A -85,B 0,C 180,E1 -2982.847,E2 -2982.847} C_VEL
LIN {X 0,Y 560.277,Z 426.721,A -85,B 0,C 180,E1 -2984.112,E2 -2984.112} C_VEL
LIN {X 0,Y 559.556,Z 421.014,A -85,B 0,C 180,E1 -2984.223,E2 -2984.223} C_VEL
LIN {X 0,Y 559.898,Z 394.253,A -85,B 0,C 180,E1 -2987.319,E2 -2987.319} C_VEL
LIN {X 0,Y 560.202,Z 371.149,A -85,B 0,C 180,E1 -2989.99,E2 -2989.99} C_VEL
LIN {X 0,Y 560.441,Z 345.628,A -85,B 0,C 180,E1 -2992.876,E2 -2992.876} C_VEL
LIN {X 0,Y 560.559,Z 320.916,A -85,B 0,C 180,E1 -2995.707,E2 -2995.707} C_VEL
LIN {X 0,Y 560.108,Z 316.377,A -85,B 0,C 180,E1 -2996.251,E2 -2996.251} C_VEL
LIN {X 0,Y 559.129,Z 311.841,A -85,B 0,C 180,E1 -2996.818,E2 -2996.818} C_VEL
LIN {X 0,Y 559.15,Z 311.834,A -85,B 0,C 180,E1 -2999.857,E2 -2999.857} C_VEL
LIN {X 0,Y 559.156,Z 311.836,A -85,B 0,C 180,E1 -3002.715,E2 -3002.715} C_VEL
LIN {X 0,Y 559.126,Z 311.834,A -85,B 0,C 180,E1 -3005.324,E2 -3005.324} C_VEL
LIN {X 0,Y 559.132,Z 311.838,A -85,B 0,C 180,E1 -3008.018,E2 -3008.018} C_VEL
LIN {X 0,Y 559.129,Z 311.835,A -85,B 0,C 180,E1 -3010.815,E2 -3010.815} C_VEL
LIN {X 0,Y 559.129,Z 311.833,A -85,B 0,C 180,E1 -3013.194,E2 -3013.194} C_VEL
LIN {X 0,Y 559.126,Z 311.837,A -85,B 0,C 180,E1 -3015.764,E2 -3015.764} C_VEL
LIN {X 0,Y 559.126,Z 311.84,A -85,B 0,C 180,E1 -3018.226,E2 -3018.226} C_VEL
LIN {X 0,Y 559.171,Z 311.828,A -85,B 0,C 180,E1 -3021.193,E2 -3021.193} C_VEL
LIN {X 0,Y 559.115,Z 311.841,A -85,B 0,C 180,E1 -3023.787,E2 -3023.787} C_VEL
LIN {X 0,Y 559.146,Z 311.832,A -85,B 0,C 180,E1 -3026.424,E2 -3026.424} C_VEL
LIN {X 0,Y 559.144,Z 311.831,A -85,B 0,C 180,E1 -3028.98,E2 -3028.98} C_VEL
LIN {X 0,Y 559.104,Z 311.844,A -85,B 0,C 180,E1 -3031.632,E2 -3031.632} C_VEL
LIN {X 0,Y 559.14,Z 311.839,A -85,B 0,C 180,E1 -3033.901,E2 -3033.901} C_VEL
LIN {X 0,Y 559.11,Z 311.838,A -85,B 0,C 180,E1 -3037.066,E2 -3037.066} C_VEL
LIN {X 0,Y 559.102,Z 311.843,A -85,B 0,C 180,E1 -3039.392,E2 -3039.392} C_VEL
LIN {X 0,Y 559.109,Z 311.843,A -85,B 0,C 180,E1 -3041.684,E2 -3041.684} C_VEL
LIN {X 0,Y 559.136,Z 311.837,A -85,B 0,C 180,E1 -3043.947,E2 -3043.947} C_VEL
LIN {X 0,Y 559.146,Z 311.834,A -85,B 0,C 180,E1 -3046.183,E2 -3046.183} C_VEL
LIN {X 0,Y 559.157,Z 311.833,A -85,B 0,C 180,E1 -3048.095,E2 -3048.095} C_VEL
LIN {X 0,Y 560.266,Z 315.731,A -85,B 0,C 180,E1 -3048.179,E2 -3048.179} C_VEL
LIN {X 0,Y 559.99,Z 400.807,A -85,B 0,C 180,E1 -3049.286,E2 -3049.286} C_VEL
LIN {X 0,Y 559.85,Z 414.004,A -85,B 0,C 180,E1 -3049.603,E2 -3049.603} C_VEL
LIN {X 0,Y 559.746,Z 426.769,A -85,B 0,C 180,E1 -3050.058,E2 -3050.058} C_VEL
LIN {X 0,Y 559.657,Z 437.941,A -85,B 0,C 180,E1 -3050.604,E2 -3050.604} C_VEL
LIN {X 0,Y 559.456,Z 448.278,A -85,B 0,C 180,E1 -3051.238,E2 -3051.238} C_VEL
LIN {X 0,Y 559.348,Z 456.813,A -85,B 0,C 180,E1 -3051.874,E2 -3051.874} C_VEL
LIN {X 0,Y 559.244,Z 464.999,A -85,B 0,C 180,E1 -3052.599,E2 -3052.599} C_VEL
LIN {X 0,Y 559.157,Z 472.308,A -85,B 0,C 180,E1 -3053.364,E2 -3053.364} C_VEL
LIN {X 0,Y 558.983,Z 479.268,A -85,B 0,C 180,E1 -3054.227,E2 -3054.227} C_VEL
LIN {X 0,Y 559.013,Z 485.367,A -85,B 0,C 180,E1 -3055.132,E2 -3055.132} C_VEL
LIN {X 0,Y 558.913,Z 490.457,A -85,B 0,C 180,E1 -3056.034,E2 -3056.034} C_VEL
LIN {X 0,Y 558.826,Z 495.379,A -85,B 0,C 180,E1 -3057.116,E2 -3057.116} C_VEL
LIN {X 0,Y 558.824,Z 499.196,A -85,B 0,C 180,E1 -3058.198,E2 -3058.198} C_VEL
LIN {X 0,Y 558.744,Z 502,A -85,B 0,C 180,E1 -3059.279,E2 -3059.279} C_VEL
LIN {X 0,Y 558.74,Z 503.39,A -85,B 0,C 180,E1 -3060,E2 -3060} C_VEL
LIN {X 0,Y 558.742,Z 504.303,A -85,B 0,C 180,E1 -3060.72,E2 -3060.72} C_VEL
LIN {X 0,Y 558.743,Z 504.981,A -85,B 0,C 180,E1 -3062.162,E2 -3062.162} C_VEL
LIN {X 0,Y 558.795,Z 504.698,A -85,B 0,C 180,E1 -3062.883,E2 -3062.883} C_VEL
LIN {X 0,Y 558.807,Z 502.998,A -85,B 0,C 180,E1 -3064.327,E2 -3064.327} C_VEL
LIN {X 0,Y 558.775,Z 501.493,A -85,B 0,C 180,E1 -3065.051,E2 -3065.051} C_VEL
LIN {X 0,Y 558.845,Z 497.24,A -85,B 0,C 180,E1 -3066.499,E2 -3066.499} C_VEL
LIN {X 0,Y 558.9,Z 492.759,A -85,B 0,C 180,E1 -3067.587,E2 -3067.587} C_VEL
LIN {X 0,Y 558.927,Z 487.047,A -85,B 0,C 180,E1 -3068.678,E2 -3068.678} C_VEL
LIN {X 0,Y 559.009,Z 481.231,A -85,B 0,C 180,E1 -3069.589,E2 -3069.589} C_VEL
LIN {X 0,Y 559.127,Z 474.226,A -85,B 0,C 180,E1 -3070.501,E2 -3070.501} C_VEL
LIN {X 0,Y 559.178,Z 467.641,A -85,B 0,C 180,E1 -3071.23,E2 -3071.23} C_VEL
LIN {X 0,Y 559.306,Z 458.717,A -85,B 0,C 180,E1 -3072.058,E2 -3072.058} C_VEL
LIN {X 0,Y 559.432,Z 450.446,A -85,B 0,C 180,E1 -3072.7,E2 -3072.7} C_VEL
LIN {X 0,Y 559.558,Z 442.021,A -85,B 0,C 180,E1 -3073.251,E2 -3073.251} C_VEL
LIN {X 0,Y 559.703,Z 431.689,A -85,B 0,C 180,E1 -3073.802,E2 -3073.802} C_VEL
LIN {X 0,Y 559.858,Z 421.931,A -85,B 0,C 180,E1 -3074.215,E2 -3074.215} C_VEL
LIN {X 0,Y 559.908,Z 411.456,A -85,B 0,C 180,E1 -3074.555,E2 -3074.555} C_VEL
LIN {X 0,Y 560.043,Z 400.173,A -85,B 0,C 180,E1 -3074.814,E2 -3074.814} C_VEL
LIN {X 0,Y 560.236,Z 315.447,A -85,B 0,C 180,E1 -3075.916,E2 -3075.916} C_VEL
LIN {X 0,Y 559.174,Z 311.83,A -85,B 0,C 180,E1 -3076.005,E2 -3076.005} C_VEL
LIN {X 0,Y 559.144,Z 311.834,A -85,B 0,C 180,E1 -3078.807,E2 -3078.807} C_VEL
LIN {X 0,Y 558.505,Z 311.915,A -85,B 0,C 180,E1 -3079.409,E2 -3079.409} C_VEL
LIN {X 0,Y 555.658,Z 312.27,A -85,B 0,C 180,E1 -3080.385,E2 -3080.385} C_VEL
LIN {X 0,Y 553.231,Z 312.57,A -85,B 0,C 180,E1 -3081.171,E2 -3081.171} C_VEL
LIN {X 0,Y 552.181,Z 312.698,A -85,B 0,C 180,E1 -3081.778,E2 -3081.778} C_VEL
LIN {X 0,Y 552.092,Z 312.71,A -85,B 0,C 180,E1 -3081.984,E2 -3081.984} C_VEL
LIN {X 0,Y 552.114,Z 312.713,A -85,B 0,C 180,E1 -3084.838,E2 -3084.838} C_VEL
LIN {X 0,Y 552.13,Z 312.705,A -85,B 0,C 180,E1 -3087.273,E2 -3087.273} C_VEL
LIN {X 0,Y 552.114,Z 312.708,A -85,B 0,C 180,E1 -3090.05,E2 -3090.05} C_VEL
LIN {X 0,Y 552.111,Z 312.712,A -85,B 0,C 180,E1 -3092.845,E2 -3092.845} C_VEL
LIN {X 0,Y 552.076,Z 312.711,A -85,B 0,C 180,E1 -3095.439,E2 -3095.439} C_VEL
LIN {X 0,Y 552.095,Z 312.71,A -85,B 0,C 180,E1 -3097.885,E2 -3097.885} C_VEL
LIN {X 0,Y 552.108,Z 312.716,A -85,B 0,C 180,E1 -3100.481,E2 -3100.481} C_VEL
LIN {X 0,Y 552.118,Z 312.706,A -85,B 0,C 180,E1 -3103.484,E2 -3103.484} C_VEL
LIN {X 0,Y 552.105,Z 312.715,A -85,B 0,C 180,E1 -3106.576,E2 -3106.576} C_VEL
LIN {X 0,Y 552.108,Z 312.707,A -85,B 0,C 180,E1 -3109.519,E2 -3109.519} C_VEL
LIN {X 0,Y 552.092,Z 312.717,A -85,B 0,C 180,E1 -3112.336,E2 -3112.336} C_VEL
LIN {X 0,Y 552.125,Z 312.706,A -85,B 0,C 180,E1 -3115.054,E2 -3115.054} C_VEL
LIN {X 0,Y 552.125,Z 312.706,A -85,B 0,C 180,E1 -3117.682,E2 -3117.682} C_VEL
LIN {X 0,Y 552.111,Z 312.715,A -85,B 0,C 180,E1 -3120.235,E2 -3120.235} C_VEL
LIN {X 0,Y 552.137,Z 312.704,A -85,B 0,C 180,E1 -3122.999,E2 -3122.999} C_VEL
LIN {X 0,Y 552.111,Z 312.707,A -85,B 0,C 180,E1 -3125.161,E2 -3125.161} C_VEL
LIN {X 0,Y 552.093,Z 312.71,A -85,B 0,C 180,E1 -3127.549,E2 -3127.549} C_VEL
LIN {X 0,Y 552.154,Z 312.704,A -85,B 0,C 180,E1 -3130.674,E2 -3130.674} C_VEL
LIN {X 0,Y 552.114,Z 312.71,A -85,B 0,C 180,E1 -3133.737,E2 -3133.737} C_VEL
LIN {X 0,Y 552.134,Z 312.711,A -85,B 0,C 180,E1 -3136.004,E2 -3136.004} C_VEL
LIN {X 0,Y 552.161,Z 312.701,A -85,B 0,C 180,E1 -3138.993,E2 -3138.993} C_VEL
LIN {X 0,Y 552.156,Z 312.708,A -85,B 0,C 180,E1 -3141.952,E2 -3141.952} C_VEL
LIN {X 0,Y 552.225,Z 312.693,A -85,B 0,C 180,E1 -3144.889,E2 -3144.889} C_VEL
LIN {X 0,Y 552.225,Z 312.699,A -85,B 0,C 180,E1 -3147.812,E2 -3147.812} C_VEL
LIN {X 0,Y 552.241,Z 312.691,A -85,B 0,C 180,E1 -3150.729,E2 -3150.729} C_VEL
LIN {X 0,Y 552.202,Z 312.695,A -85,B 0,C 180,E1 -3152.918,E2 -3152.918} C_VEL
LIN {X 0,Y 552.198,Z 312.703,A -85,B 0,C 180,E1 -3155.844,E2 -3155.844} C_VEL
LIN {X 0,Y 552.156,Z 312.701,A -85,B 0,C 180,E1 -3158.786,E2 -3158.786} C_VEL
LIN {X 0,Y 552.161,Z 312.707,A -85,B 0,C 180,E1 -3161.751,E2 -3161.751} C_VEL
LIN {X 0,Y 552.135,Z 312.704,A -85,B 0,C 180,E1 -3164.749,E2 -3164.749} C_VEL
LIN {X 0,Y 552.112,Z 312.715,A -85,B 0,C 180,E1 -3167.789,E2 -3167.789} C_VEL
LIN {X 0,Y 552.129,Z 312.71,A -85,B 0,C 180,E1 -3170.102,E2 -3170.102} C_VEL
LIN {X 0,Y 552.094,Z 312.71,A -85,B 0,C 180,E1 -3172.451,E2 -3172.451} C_VEL
LIN {X 0,Y 552.155,Z 312.705,A -85,B 0,C 180,E1 -3175.351,E2 -3175.351} C_VEL
LIN {X 0,Y 552.119,Z 312.71,A -85,B 0,C 180,E1 -3178.098,E2 -3178.098} C_VEL
LIN {X 0,Y 552.107,Z 312.707,A -85,B 0,C 180,E1 -3180.609,E2 -3180.609} C_VEL
LIN {X 0,Y 552.123,Z 312.708,A -85,B 0,C 180,E1 -3183.186,E2 -3183.186} C_VEL
LIN {X 0,Y 552.103,Z 312.715,A -85,B 0,C 180,E1 -3185.843,E2 -3185.843} C_VEL
LIN {X 0,Y 552.125,Z 312.707,A -85,B 0,C 180,E1 -3189.062,E2 -3189.062} C_VEL
LIN {X 0,Y 552.121,Z 312.712,A -85,B 0,C 180,E1 -3191.446,E2 -3191.446} C_VEL
LIN {X 0,Y 552.091,Z 312.709,A -85,B 0,C 180,E1 -3194.532,E2 -3194.532} C_VEL
LIN {X 0,Y 552.13,Z 312.713,A -85,B 0,C 180,E1 -3197.585,E2 -3197.585} C_VEL
LIN {X 0,Y 552.13,Z 312.704,A -85,B 0,C 180,E1 -3200.473,E2 -3200.473} C_VEL
LIN {X 0,Y 552.108,Z 312.714,A -85,B 0,C 180,E1 -3203.318,E2 -3203.318} C_VEL
LIN {X 0,Y 552.105,Z 312.711,A -85,B 0,C 180,E1 -3205.938,E2 -3205.938} C_VEL
LIN {X 0,Y 552.122,Z 312.706,A -85,B 0,C 180,E1 -3208.541,E2 -3208.541} C_VEL
LIN {X 0,Y 552.127,Z 312.713,A -85,B 0,C 180,E1 -3211.439,E2 -3211.439} C_VEL
LIN {X 0,Y 552.131,Z 312.704,A -85,B 0,C 180,E1 -3214.356,E2 -3214.356} C_VEL
LIN {X 0,Y 552.098,Z 312.711,A -85,B 0,C 180,E1 -3216.758,E2 -3216.758} C_VEL
LIN {X 0,Y 552.128,Z 312.71,A -85,B 0,C 180,E1 -3217.923,E2 -3217.923} C_VEL
LIN {X 0,Y 553.386,Z 317.783,A -85,B 0,C 180,E1 -3218.029,E2 -3218.029} C_VEL
LIN {X 0,Y 553.118,Z 399.504,A -85,B 0,C 180,E1 -3219.111,E2 -3219.111} C_VEL
LIN {X 0,Y 553.034,Z 409.568,A -85,B 0,C 180,E1 -3219.327,E2 -3219.327} C_VEL
LIN {X 0,Y 552.913,Z 418.385,A -85,B 0,C 180,E1 -3219.589,E2 -3219.589} C_VEL
LIN {X 0,Y 552.787,Z 429.264,A -85,B 0,C 180,E1 -3220.024,E2 -3220.024} C_VEL
LIN {X 0,Y 552.663,Z 438.839,A -85,B 0,C 180,E1 -3220.512,E2 -3220.512} C_VEL
LIN {X 0,Y 552.495,Z 447.864,A -85,B 0,C 180,E1 -3221.073,E2 -3221.073} C_VEL
LIN {X 0,Y 552.313,Z 456.755,A -85,B 0,C 180,E1 -3221.739,E2 -3221.739} C_VEL
LIN {X 0,Y 552.24,Z 463.914,A -85,B 0,C 180,E1 -3222.371,E2 -3222.371} C_VEL
LIN {X 0,Y 552.097,Z 471.567,A -85,B 0,C 180,E1 -3223.166,E2 -3223.166} C_VEL
LIN {X 0,Y 551.965,Z 479.151,A -85,B 0,C 180,E1 -3224.113,E2 -3224.113} C_VEL
LIN {X 0,Y 551.868,Z 485.437,A -85,B 0,C 180,E1 -3225.056,E2 -3225.056} C_VEL
LIN {X 0,Y 551.805,Z 490.639,A -85,B 0,C 180,E1 -3225.996,E2 -3225.996} C_VEL
LIN {X 0,Y 551.739,Z 495.631,A -85,B 0,C 180,E1 -3227.12,E2 -3227.12} C_VEL
LIN {X 0,Y 551.732,Z 499.46,A -85,B 0,C 180,E1 -3228.241,E2 -3228.241} C_VEL
LIN {X 0,Y 551.705,Z 501.452,A -85,B 0,C 180,E1 -3228.985,E2 -3228.985} C_VEL
LIN {X 0,Y 551.677,Z 502.987,A -85,B 0,C 180,E1 -3229.727,E2 -3229.727} C_VEL
LIN {X 0,Y 551.671,Z 504.694,A -85,B 0,C 180,E1 -3231.207,E2 -3231.207} C_VEL
LIN {X 0,Y 551.696,Z 504.985,A -85,B 0,C 180,E1 -3231.945,E2 -3231.945} C_VEL
LIN {X 0,Y 551.731,Z 504.151,A -85,B 0,C 180,E1 -3233.504,E2 -3233.504} C_VEL
LIN {X 0,Y 551.713,Z 503.34,A -85,B 0,C 180,E1 -3234.151,E2 -3234.151} C_VEL
LIN {X 0,Y 551.722,Z 500.147,A -85,B 0,C 180,E1 -3235.617,E2 -3235.617} C_VEL
LIN {X 0,Y 551.78,Z 496.619,A -85,B 0,C 180,E1 -3236.715,E2 -3236.715} C_VEL
LIN {X 0,Y 551.734,Z 492.017,A -85,B 0,C 180,E1 -3237.81,E2 -3237.81} C_VEL
LIN {X 0,Y 551.871,Z 486.196,A -85,B 0,C 180,E1 -3238.906,E2 -3238.906} C_VEL
LIN {X 0,Y 551.965,Z 480.282,A -85,B 0,C 180,E1 -3239.818,E2 -3239.818} C_VEL
LIN {X 0,Y 552.064,Z 473.205,A -85,B 0,C 180,E1 -3240.73,E2 -3240.73} C_VEL
LIN {X 0,Y 552.172,Z 466.52,A -85,B 0,C 180,E1 -3241.459,E2 -3241.459} C_VEL
LIN {X 0,Y 552.306,Z 458.678,A -85,B 0,C 180,E1 -3242.188,E2 -3242.188} C_VEL
LIN {X 0,Y 552.44,Z 450.578,A -85,B 0,C 180,E1 -3242.826,E2 -3242.826} C_VEL
LIN {X 0,Y 552.619,Z 442.369,A -85,B 0,C 180,E1 -3243.372,E2 -3243.372} C_VEL
LIN {X 0,Y 552.784,Z 432.364,A -85,B 0,C 180,E1 -3243.919,E2 -3243.919} C_VEL
LIN {X 0,Y 552.857,Z 421.83,A -85,B 0,C 180,E1 -3244.375,E2 -3244.375} C_VEL
LIN {X 0,Y 552.962,Z 412.207,A -85,B 0,C 180,E1 -3244.693,E2 -3244.693} C_VEL
LIN {X 0,Y 553.048,Z 401.587,A -85,B 0,C 180,E1 -3244.944,E2 -3244.944} C_VEL
LIN {X 0,Y 553.168,Z 375.645,A -85,B 0,C 180,E1 -3245.308,E2 -3245.308} C_VEL
LIN {X 0,Y 553.277,Z 316.58,A -85,B 0,C 180,E1 -3246.081,E2 -3246.081} C_VEL
LIN {X 0,Y 552.12,Z 312.711,A -85,B 0,C 180,E1 -3246.166,E2 -3246.166} C_VEL
LIN {X 0,Y 552.128,Z 312.714,A -85,B 0,C 180,E1 -3248.786,E2 -3248.786} C_VEL
LIN {X 0,Y 552.084,Z 312.712,A -85,B 0,C 180,E1 -3251.753,E2 -3251.753} C_VEL
LIN {X 0,Y 552.126,Z 312.712,A -85,B 0,C 180,E1 -3254.749,E2 -3254.749} C_VEL
LIN {X 0,Y 552.08,Z 312.713,A -85,B 0,C 180,E1 -3257.79,E2 -3257.79} C_VEL
LIN {X 0,Y 552.051,Z 312.721,A -85,B 0,C 180,E1 -3260.105,E2 -3260.105} C_VEL
LIN {X 0,Y 552.054,Z 312.721,A -85,B 0,C 180,E1 -3262.453,E2 -3262.453} C_VEL
LIN {X 0,Y 552.074,Z 312.712,A -85,B 0,C 180,E1 -3265.331,E2 -3265.331} C_VEL
LIN {X 0,Y 552.051,Z 312.722,A -85,B 0,C 180,E1 -3268.102,E2 -3268.102} C_VEL
LIN {X 0,Y 552.09,Z 312.713,A -85,B 0,C 180,E1 -3270.61,E2 -3270.61} C_VEL
LIN {X 0,Y 552.108,Z 312.707,A -85,B 0,C 180,E1 -3273.187,E2 -3273.187} C_VEL
LIN {X 0,Y 552.072,Z 312.717,A -85,B 0,C 180,E1 -3275.845,E2 -3275.845} C_VEL
LIN {X 0,Y 552.115,Z 312.707,A -85,B 0,C 180,E1 -3278.59,E2 -3278.59} C_VEL
LIN {X 0,Y 552.073,Z 312.713,A -85,B 0,C 180,E1 -3281.451,E2 -3281.451} C_VEL
LIN {X 0,Y 552.079,Z 312.712,A -85,B 0,C 180,E1 -3284.529,E2 -3284.529} C_VEL
LIN {X 0,Y 552.112,Z 312.713,A -85,B 0,C 180,E1 -3287.587,E2 -3287.587} C_VEL
LIN {X 0,Y 552.131,Z 312.705,A -85,B 0,C 180,E1 -3290.472,E2 -3290.472} C_VEL
LIN {X 0,Y 552.101,Z 312.713,A -85,B 0,C 180,E1 -3293.318,E2 -3293.318} C_VEL
LIN {X 0,Y 552.121,Z 312.71,A -85,B 0,C 180,E1 -3295.938,E2 -3295.938} C_VEL
LIN {X 0,Y 552.124,Z 312.706,A -85,B 0,C 180,E1 -3298.541,E2 -3298.541} C_VEL
LIN {X 0,Y 552.102,Z 312.717,A -85,B 0,C 180,E1 -3301.443,E2 -3301.443} C_VEL
LIN {X 0,Y 552.154,Z 312.904,A -85,B 0,C 180,E1 -3302.814,E2 -3302.814} C_VEL
LIN {X 0,Y 553.951,Z 322.139,A -85,B 0,C 180,E1 -3304.01,E2 -3304.01} C_VEL
LIN {X 0,Y 553.652,Z 344.079,A -85,B 0,C 180,E1 -3306.629,E2 -3306.629} C_VEL
LIN {X 0,Y 553.275,Z 368.864,A -85,B 0,C 180,E1 -3309.554,E2 -3309.554} C_VEL
LIN {X 0,Y 552.954,Z 394.819,A -85,B 0,C 180,E1 -3312.543,E2 -3312.543} C_VEL
LIN {X 0,Y 552.591,Z 421.336,A -85,B 0,C 180,E1 -3315.617,E2 -3315.617} C_VEL
LIN {X 0,Y 553.481,Z 428.491,A -85,B 0,C 180,E1 -3315.734,E2 -3315.734} C_VEL
LIN {X 0,Y 553.112,Z 530.935,A -85,B 0,C 180,E1 -3317.082,E2 -3317.082} C_VEL
LIN {X 0,Y 552.985,Z 544.21,A -85,B 0,C 180,E1 -3317.406,E2 -3317.406} C_VEL
LIN {X 0,Y 552.808,Z 557.483,A -85,B 0,C 180,E1 -3317.891,E2 -3317.891} C_VEL
LIN {X 0,Y 552.631,Z 569.195,A -85,B 0,C 180,E1 -3318.479,E2 -3318.479} C_VEL
LIN {X 0,Y 552.456,Z 581.483,A -85,B 0,C 180,E1 -3319.277,E2 -3319.277} C_VEL
LIN {X 0,Y 552.277,Z 591.644,A -85,B 0,C 180,E1 -3320.108,E2 -3320.108} C_VEL
LIN {X 0,Y 552.104,Z 600.784,A -85,B 0,C 180,E1 -3321.029,E2 -3321.029} C_VEL
LIN {X 0,Y 551.96,Z 609.687,A -85,B 0,C 180,E1 -3322.133,E2 -3322.133} C_VEL
LIN {X 0,Y 551.836,Z 616.848,A -85,B 0,C 180,E1 -3323.234,E2 -3323.234} C_VEL
LIN {X 0,Y 551.804,Z 623.365,A -85,B 0,C 180,E1 -3324.518,E2 -3324.518} C_VEL
LIN {X 0,Y 551.764,Z 627.676,A -85,B 0,C 180,E1 -3325.617,E2 -3325.617} C_VEL
LIN {X 0,Y 551.75,Z 629.958,A -85,B 0,C 180,E1 -3326.348,E2 -3326.348} C_VEL
LIN {X 0,Y 551.724,Z 631.807,A -85,B 0,C 180,E1 -3327.079,E2 -3327.079} C_VEL
LIN {X 0,Y 551.645,Z 634.183,A -85,B 0,C 180,E1 -3328.54,E2 -3328.54} C_VEL
LIN {X 0,Y 551.64,Z 635,A -85,B 0,C 180,E1 -3330,E2 -3330} C_VEL
LIN {X 0,Y 551.645,Z 634.185,A -85,B 0,C 180,E1 -3331.46,E2 -3331.46} C_VEL
LIN {X 0,Y 551.724,Z 631.81,A -85,B 0,C 180,E1 -3332.921,E2 -3332.921} C_VEL
LIN {X 0,Y 551.764,Z 628.896,A -85,B 0,C 180,E1 -3334.017,E2 -3334.017} C_VEL
LIN {X 0,Y 551.724,Z 624.949,A -85,B 0,C 180,E1 -3335.116,E2 -3335.116} C_VEL
LIN {X 0,Y 551.815,Z 619.125,A -85,B 0,C 180,E1 -3336.353,E2 -3336.353} C_VEL
LIN {X 0,Y 551.927,Z 612.237,A -85,B 0,C 180,E1 -3337.5,E2 -3337.5} C_VEL
LIN {X 0,Y 552.082,Z 603.992,A -85,B 0,C 180,E1 -3338.602,E2 -3338.602} C_VEL
LIN {X 0,Y 552.221,Z 595.54,A -85,B 0,C 180,E1 -3339.523,E2 -3339.523} C_VEL
LIN {X 0,Y 552.432,Z 585.094,A -85,B 0,C 180,E1 -3340.445,E2 -3340.445} C_VEL
LIN {X 0,Y 552.556,Z 574.288,A -85,B 0,C 180,E1 -3341.214,E2 -3341.214} C_VEL
LIN {X 0,Y 552.782,Z 563.406,A -85,B 0,C 180,E1 -3341.83,E2 -3341.83} C_VEL
LIN {X 0,Y 552.877,Z 551.765,A -85,B 0,C 180,E1 -3342.34,E2 -3342.34} C_VEL
LIN {X 0,Y 553.074,Z 538.346,A -85,B 0,C 180,E1 -3342.755,E2 -3342.755} C_VEL
LIN {X 0,Y 553.147,Z 525.086,A -85,B 0,C 180,E1 -3343.01,E2 -3343.01} C_VEL
LIN {X 0,Y 553.329,Z 426.721,A -85,B 0,C 180,E1 -3344.293,E2 -3344.293} C_VEL
LIN {X 0,Y 552.59,Z 421.014,A -85,B 0,C 180,E1 -3344.407,E2 -3344.407} C_VEL
LIN {X 0,Y 552.94,Z 394.775,A -85,B 0,C 180,E1 -3347.46,E2 -3347.46} C_VEL
LIN {X 0,Y 553.25,Z 366.663,A -85,B 0,C 180,E1 -3350.641,E2 -3350.641} C_VEL
LIN {X 0,Y 553.461,Z 342.898,A -85,B 0,C 180,E1 -3353.377,E2 -3353.377} C_VEL
LIN {X 0,Y 553.601,Z 320.574,A -85,B 0,C 180,E1 -3355.975,E2 -3355.975} C_VEL
LIN {X 0,Y 552.086,Z 312.717,A -85,B 0,C 180,E1 -3356.989,E2 -3356.989} C_VEL
LIN {X 0,Y 552.119,Z 312.712,A -85,B 0,C 180,E1 -3360.05,E2 -3360.05} C_VEL
LIN {X 0,Y 552.114,Z 312.712,A -85,B 0,C 180,E1 -3362.846,E2 -3362.846} C_VEL
LIN {X 0,Y 552.073,Z 312.713,A -85,B 0,C 180,E1 -3365.439,E2 -3365.439} C_VEL
LIN {X 0,Y 552.095,Z 312.713,A -85,B 0,C 180,E1 -3367.885,E2 -3367.885} C_VEL
LIN {X 0,Y 552.095,Z 312.716,A -85,B 0,C 180,E1 -3370.483,E2 -3370.483} C_VEL
LIN {X 0,Y 552.095,Z 312.711,A -85,B 0,C 180,E1 -3373.481,E2 -3373.481} C_VEL
LIN {X 0,Y 552.075,Z 312.714,A -85,B 0,C 180,E1 -3376.573,E2 -3376.573} C_VEL
LIN {X 0,Y 552.094,Z 312.711,A -85,B 0,C 180,E1 -3379.517,E2 -3379.517} C_VEL
LIN {X 0,Y 552.084,Z 312.714,A -85,B 0,C 180,E1 -3382.335,E2 -3382.335} C_VEL
LIN {X 0,Y 552.073,Z 312.712,A -85,B 0,C 180,E1 -3385.05,E2 -3385.05} C_VEL
LIN {X 0,Y 552.106,Z 312.714,A -85,B 0,C 180,E1 -3387.68,E2 -3387.68} C_VEL
LIN {X 0,Y 552.073,Z 312.715,A -85,B 0,C 180,E1 -3390.232,E2 -3390.232} C_VEL
LIN {X 0,Y 552.076,Z 312.712,A -85,B 0,C 180,E1 -3393.013,E2 -3393.013} C_VEL
LIN {X 0,Y 552.075,Z 312.718,A -85,B 0,C 180,E1 -3395.96,E2 -3395.96} C_VEL
LIN {X 0,Y 552.059,Z 312.717,A -85,B 0,C 180,E1 -3399.117,E2 -3399.117} C_VEL
LIN {X 0,Y 552.068,Z 312.721,A -85,B 0,C 180,E1 -3401.442,E2 -3401.442} C_VEL
LIN {X 0,Y 552.084,Z 312.718,A -85,B 0,C 180,E1 -3403.736,E2 -3403.736} C_VEL
LIN {X 0,Y 552.114,Z 312.711,A -85,B 0,C 180,E1 -3406.004,E2 -3406.004} C_VEL
LIN {X 0,Y 552.13,Z 312.71,A -85,B 0,C 180,E1 -3407.908,E2 -3407.908} C_VEL
LIN {X 0,Y 553.363,Z 317.182,A -85,B 0,C 180,E1 -3408.019,E2 -3408.019} C_VEL
LIN {X 0,Y 553.087,Z 400.973,A -85,B 0,C 180,E1 -3409.128,E2 -3409.128} C_VEL
LIN {X 0,Y 552.941,Z 413.251,A -85,B 0,C 180,E1 -3409.426,E2 -3409.426} C_VEL
LIN {X 0,Y 552.81,Z 426.319,A -85,B 0,C 180,E1 -3409.886,E2 -3409.886} C_VEL
LIN {X 0,Y 552.678,Z 438.378,A -85,B 0,C 180,E1 -3410.484,E2 -3410.484} C_VEL
LIN {X 0,Y 552.521,Z 447.34,A -85,B 0,C 180,E1 -3411.035,E2 -3411.035} C_VEL
LIN {X 0,Y 552.323,Z 457.112,A -85,B 0,C 180,E1 -3411.77,E2 -3411.77} C_VEL
LIN {X 0,Y 552.203,Z 465.25,A -85,B 0,C 180,E1 -3412.504,E2 -3412.504} C_VEL
LIN {X 0,Y 552.075,Z 471.824,A -85,B 0,C 180,E1 -3413.196,E2 -3413.196} C_VEL
LIN {X 0,Y 551.933,Z 479.443,A -85,B 0,C 180,E1 -3414.153,E2 -3414.153} C_VEL
LIN {X 0,Y 551.948,Z 485.512,A -85,B 0,C 180,E1 -3415.069,E2 -3415.069} C_VEL
LIN {X 0,Y 551.826,Z 490.575,A -85,B 0,C 180,E1 -3415.983,E2 -3415.983} C_VEL
LIN {X 0,Y 551.752,Z 495.473,A -85,B 0,C 180,E1 -3417.079,E2 -3417.079} C_VEL
LIN {X 0,Y 551.743,Z 499.265,A -85,B 0,C 180,E1 -3418.175,E2 -3418.175} C_VEL
LIN {X 0,Y 551.645,Z 502.045,A -85,B 0,C 180,E1 -3419.27,E2 -3419.27} C_VEL
LIN {X 0,Y 551.641,Z 503.425,A -85,B 0,C 180,E1 -3420,E2 -3420} C_VEL
LIN {X 0,Y 551.643,Z 504.326,A -85,B 0,C 180,E1 -3420.73,E2 -3420.73} C_VEL
LIN {X 0,Y 551.654,Z 504.975,A -85,B 0,C 180,E1 -3422.19,E2 -3422.19} C_VEL
LIN {X 0,Y 551.719,Z 504.678,A -85,B 0,C 180,E1 -3422.92,E2 -3422.92} C_VEL
LIN {X 0,Y 551.702,Z 502.943,A -85,B 0,C 180,E1 -3424.383,E2 -3424.383} C_VEL
LIN {X 0,Y 551.694,Z 501.429,A -85,B 0,C 180,E1 -3425.116,E2 -3425.116} C_VEL
LIN {X 0,Y 551.768,Z 497.031,A -85,B 0,C 180,E1 -3426.608,E2 -3426.608} C_VEL
LIN {X 0,Y 551.81,Z 492.62,A -85,B 0,C 180,E1 -3427.685,E2 -3427.685} C_VEL
LIN {X 0,Y 551.853,Z 486.879,A -85,B 0,C 180,E1 -3428.79,E2 -3428.79} C_VEL
LIN {X 0,Y 551.949,Z 481.029,A -85,B 0,C 180,E1 -3429.713,E2 -3429.713} C_VEL
LIN {X 0,Y 552.052,Z 475.548,A -85,B 0,C 180,E1 -3430.452,E2 -3430.452} C_VEL
LIN {X 0,Y 552.142,Z 468.132,A -85,B 0,C 180,E1 -3431.298,E2 -3431.298} C_VEL
LIN {X 0,Y 552.27,Z 459.483,A -85,B 0,C 180,E1 -3432.12,E2 -3432.12} C_VEL
LIN {X 0,Y 552.414,Z 451.364,A -85,B 0,C 180,E1 -3432.77,E2 -3432.77} C_VEL
LIN {X 0,Y 552.585,Z 441.544,A -85,B 0,C 180,E1 -3433.421,E2 -3433.421} C_VEL
LIN {X 0,Y 552.728,Z 433.073,A -85,B 0,C 180,E1 -3433.886,E2 -3433.886} C_VEL
LIN {X 0,Y 552.918,Z 422.439,A -85,B 0,C 180,E1 -3434.35,E2 -3434.35} C_VEL
LIN {X 0,Y 552.983,Z 411.885,A -85,B 0,C 180,E1 -3434.701,E2 -3434.701} C_VEL
LIN {X 0,Y 553.127,Z 399.859,A -85,B 0,C 180,E1 -3434.982,E2 -3434.982} C_VEL
LIN {X 0,Y 553.335,Z 316.78,A -85,B 0,C 180,E1 -3436.077,E2 -3436.077} C_VEL
LIN {X 0,Y 552.133,Z 312.709,A -85,B 0,C 180,E1 -3436.169,E2 -3436.169} C_VEL
LIN {X 0,Y 552.152,Z 312.703,A -85,B 0,C 180,E1 -3439.325,E2 -3439.325} C_VEL
LIN {X 0,Y 552.092,Z 312.71,A -85,B 0,C 180,E1 -3441.984,E2 -3441.984} C_VEL
LIN {X 0,Y 551.432,Z 312.8,A -85,B 0,C 180,E1 -3442.592,E2 -3442.592} C_VEL
LIN {X 0,Y 548.633,Z 313.148,A -85,B 0,C 180,E1 -3443.581,E2 -3443.581} C_VEL
LIN {X 0,Y 546.256,Z 313.443,A -85,B 0,C 180,E1 -3444.377,E2 -3444.377} C_VEL
LIN {X 0,Y 545.213,Z 313.571,A -85,B 0,C 180,E1 -3444.99,E2 -3444.99} C_VEL
LIN {X 0,Y 545.116,Z 313.58,A -85,B 0,C 180,E1 -3445.198,E2 -3445.198} C_VEL
LIN {X 0,Y 545.081,Z 313.582,A -85,B 0,C 180,E1 -3447.656,E2 -3447.656} C_VEL
LIN {X 0,Y 545.058,Z 313.589,A -85,B 0,C 180,E1 -3450.242,E2 -3450.242} C_VEL
LIN {X 0,Y 545.074,Z 313.586,A -85,B 0,C 180,E1 -3453.061,E2 -3453.061} C_VEL
LIN {X 0,Y 545.033,Z 313.588,A -85,B 0,C 180,E1 -3455.672,E2 -3455.672} C_VEL
LIN {X 0,Y 545.051,Z 313.591,A -85,B 0,C 180,E1 -3458.237,E2 -3458.237} C_VEL
LIN {X 0,Y 545.08,Z 313.591,A -85,B 0,C 180,E1 -3460.472,E2 -3460.472} C_VEL
LIN {X 0,Y 545.077,Z 313.584,A -85,B 0,C 180,E1 -3463.106,E2 -3463.106} C_VEL
LIN {X 0,Y 545.048,Z 313.593,A -85,B 0,C 180,E1 -3466.226,E2 -3466.226} C_VEL
LIN {X 0,Y 545.08,Z 313.585,A -85,B 0,C 180,E1 -3468.885,E2 -3468.885} C_VEL
LIN {X 0,Y 545.082,Z 313.586,A -85,B 0,C 180,E1 -3470.818,E2 -3470.818} C_VEL
LIN {X 0,Y 545.049,Z 313.587,A -85,B 0,C 180,E1 -3473.62,E2 -3473.62} C_VEL
LIN {X 0,Y 545.07,Z 313.592,A -85,B 0,C 180,E1 -3476.328,E2 -3476.328} C_VEL
LIN {X 0,Y 545.066,Z 313.586,A -85,B 0,C 180,E1 -3478.952,E2 -3478.952} C_VEL
LIN {X 0,Y 545.1,Z 313.581,A -85,B 0,C 180,E1 -3481.508,E2 -3481.508} C_VEL
LIN {X 0,Y 545.094,Z 313.587,A -85,B 0,C 180,E1 -3484.491,E2 -3484.491} C_VEL
LIN {X 0,Y 545.042,Z 313.587,A -85,B 0,C 180,E1 -3487.242,E2 -3487.242} C_VEL
LIN {X 0,Y 545.118,Z 313.584,A -85,B 0,C 180,E1 -3490.415,E2 -3490.415} C_VEL
LIN {X 0,Y 545.071,Z 313.585,A -85,B 0,C 180,E1 -3493.521,E2 -3493.521} C_VEL
LIN {X 0,Y 545.093,Z 313.586,A -85,B 0,C 180,E1 -3495.82,E2 -3495.82} C_VEL
LIN {X 0,Y 545.116,Z 313.579,A -85,B 0,C 180,E1 -3498.849,E2 -3498.849} C_VEL
LIN {X 0,Y 545.126,Z 313.583,A -85,B 0,C 180,E1 -3501.847,E2 -3501.847} C_VEL
LIN {X 0,Y 545.201,Z 313.568,A -85,B 0,C 180,E1 -3504.823,E2 -3504.823} C_VEL
LIN {X 0,Y 545.196,Z 313.574,A -85,B 0,C 180,E1 -3507.784,E2 -3507.784} C_VEL
LIN {X 0,Y 545.211,Z 313.567,A -85,B 0,C 180,E1 -3510.739,E2 -3510.739} C_VEL
LIN {X 0,Y 545.169,Z 313.572,A -85,B 0,C 180,E1 -3512.956,E2 -3512.956} C_VEL
LIN {X 0,Y 545.169,Z 313.579,A -85,B 0,C 180,E1 -3515.92,E2 -3515.92} C_VEL
LIN {X 0,Y 545.115,Z 313.578,A -85,B 0,C 180,E1 -3518.9,E2 -3518.9} C_VEL
LIN {X 0,Y 545.133,Z 313.584,A -85,B 0,C 180,E1 -3521.904,E2 -3521.904} C_VEL
LIN {X 0,Y 545.084,Z 313.582,A -85,B 0,C 180,E1 -3524.944,E2 -3524.944} C_VEL
LIN {X 0,Y 545.08,Z 313.59,A -85,B 0,C 180,E1 -3528.026,E2 -3528.026} C_VEL
LIN {X 0,Y 545.094,Z 313.583,A -85,B 0,C 180,E1 -3530.372,E2 -3530.372} C_VEL
LIN {X 0,Y 545.09,Z 313.587,A -85,B 0,C 180,E1 -3533.559,E2 -3533.559} C_VEL
LIN {X 0,Y 545.079,Z 313.589,A -85,B 0,C 180,E1 -3536.001,E2 -3536.001} C_VEL
LIN {X 0,Y 545.088,Z 313.582,A -85,B 0,C 180,E1 -3538.749,E2 -3538.749} C_VEL
LIN {X 0,Y 545.059,Z 313.593,A -85,B 0,C 180,E1 -3541.68,E2 -3541.68} C_VEL
LIN {X 0,Y 545.08,Z 313.583,A -85,B 0,C 180,E1 -3544.564,E2 -3544.564} C_VEL
LIN {X 0,Y 545.038,Z 313.592,A -85,B 0,C 180,E1 -3547.304,E2 -3547.304} C_VEL
LIN {X 0,Y 545.068,Z 313.587,A -85,B 0,C 180,E1 -3550.143,E2 -3550.143} C_VEL
LIN {X 0,Y 545.078,Z 313.586,A -85,B 0,C 180,E1 -3553.107,E2 -3553.107} C_VEL
LIN {X 0,Y 545.068,Z 313.586,A -85,B 0,C 180,E1 -3556.225,E2 -3556.225} C_VEL
LIN {X 0,Y 545.082,Z 313.584,A -85,B 0,C 180,E1 -3558.886,E2 -3558.886} C_VEL
LIN {X 0,Y 545.053,Z 313.592,A -85,B 0,C 180,E1 -3561.763,E2 -3561.763} C_VEL
LIN {X 0,Y 545.038,Z 313.588,A -85,B 0,C 180,E1 -3564.532,E2 -3564.532} C_VEL
LIN {X 0,Y 545.067,Z 313.59,A -85,B 0,C 180,E1 -3567.212,E2 -3567.212} C_VEL
LIN {X 0,Y 545.063,Z 313.589,A -85,B 0,C 180,E1 -3569.811,E2 -3569.811} C_VEL
LIN {X 0,Y 545.077,Z 313.583,A -85,B 0,C 180,E1 -3572.344,E2 -3572.344} C_VEL
LIN {X 0,Y 545.109,Z 313.581,A -85,B 0,C 180,E1 -3574.82,E2 -3574.82} C_VEL
LIN {X 0,Y 545.081,Z 313.611,A -85,B 0,C 180,E1 -3577.754,E2 -3577.754} C_VEL
LIN {X 0,Y 546.505,Z 319.03,A -85,B 0,C 180,E1 -3577.865,E2 -3577.865} C_VEL
LIN {X 0,Y 546.2,Z 400.181,A -85,B 0,C 180,E1 -3578.957,E2 -3578.957} C_VEL
LIN {X 0,Y 546.112,Z 410.263,A -85,B 0,C 180,E1 -3579.176,E2 -3579.176} C_VEL
LIN {X 0,Y 546.003,Z 419.739,A -85,B 0,C 180,E1 -3579.467,E2 -3579.467} C_VEL
LIN {X 0,Y 545.82,Z 430.655,A -85,B 0,C 180,E1 -3579.917,E2 -3579.917} C_VEL
LIN {X 0,Y 545.682,Z 440.474,A -85,B 0,C 180,E1 -3580.436,E2 -3580.436} C_VEL
LIN {X 0,Y 545.506,Z 449.417,A -85,B 0,C 180,E1 -3581.016,E2 -3581.016} C_VEL
LIN {X 0,Y 545.322,Z 458.06,A -85,B 0,C 180,E1 -3581.691,E2 -3581.691} C_VEL
LIN {X 0,Y 545.19,Z 466.041,A -85,B 0,C 180,E1 -3582.437,E2 -3582.437} C_VEL
LIN {X 0,Y 545.053,Z 472.434,A -85,B 0,C 180,E1 -3583.135,E2 -3583.135} C_VEL
LIN {X 0,Y 544.937,Z 478.481,A -85,B 0,C 180,E1 -3583.902,E2 -3583.902} C_VEL
LIN {X 0,Y 544.832,Z 484.803,A -85,B 0,C 180,E1 -3584.858,E2 -3584.858} C_VEL
LIN {X 0,Y 544.752,Z 490.12,A -85,B 0,C 180,E1 -3585.811,E2 -3585.811} C_VEL
LIN {X 0,Y 544.652,Z 495.218,A -85,B 0,C 180,E1 -3586.95,E2 -3586.95} C_VEL
LIN {X 0,Y 544.645,Z 499.144,A -85,B 0,C 180,E1 -3588.085,E2 -3588.085} C_VEL
LIN {X 0,Y 544.612,Z 501.227,A -85,B 0,C 180,E1 -3588.839,E2 -3588.839} C_VEL
LIN {X 0,Y 544.581,Z 502.772,A -85,B 0,C 180,E1 -3589.591,E2 -3589.591} C_VEL
LIN {X 0,Y 544.564,Z 504.643,A -85,B 0,C 180,E1 -3591.091,E2 -3591.091} C_VEL
LIN {X 0,Y 544.612,Z 504.946,A -85,B 0,C 180,E1 -3591.84,E2 -3591.84} C_VEL
LIN {X 0,Y 544.652,Z 504.375,A -85,B 0,C 180,E1 -3593.331,E2 -3593.331} C_VEL
LIN {X 0,Y 544.616,Z 503.467,A -85,B 0,C 180,E1 -3594.075,E2 -3594.075} C_VEL
LIN {X 0,Y 544.617,Z 500.442,A -85,B 0,C 180,E1 -3595.56,E2 -3595.56} C_VEL
LIN {X 0,Y 544.706,Z 497.007,A -85,B 0,C 180,E1 -3596.672,E2 -3596.672} C_VEL
LIN {X 0,Y 544.646,Z 492.506,A -85,B 0,C 180,E1 -3597.782,E2 -3597.782} C_VEL
LIN {X 0,Y 544.727,Z 487.876,A -85,B 0,C 180,E1 -3598.707,E2 -3598.707} C_VEL
LIN {X 0,Y 544.912,Z 481.063,A -85,B 0,C 180,E1 -3599.816,E2 -3599.816} C_VEL
LIN {X 0,Y 544.964,Z 475.762,A -85,B 0,C 180,E1 -3600.555,E2 -3600.555} C_VEL
LIN {X 0,Y 545.138,Z 467.806,A -85,B 0,C 180,E1 -3601.478,E2 -3601.478} C_VEL
LIN {X 0,Y 545.337,Z 459.163,A -85,B 0,C 180,E1 -3602.308,E2 -3602.308} C_VEL
LIN {X 0,Y 545.492,Z 451.149,A -85,B 0,C 180,E1 -3602.954,E2 -3602.954} C_VEL
LIN {X 0,Y 545.68,Z 443.004,A -85,B 0,C 180,E1 -3603.508,E2 -3603.508} C_VEL
LIN {X 0,Y 545.85,Z 433.051,A -85,B 0,C 180,E1 -3604.061,E2 -3604.061} C_VEL
LIN {X 0,Y 545.937,Z 422.535,A -85,B 0,C 180,E1 -3604.523,E2 -3604.523} C_VEL
LIN {X 0,Y 546.079,Z 412.014,A -85,B 0,C 180,E1 -3604.868,E2 -3604.868} C_VEL
LIN {X 0,Y 546.15,Z 402.109,A -85,B 0,C 180,E1 -3605.099,E2 -3605.099} C_VEL
LIN {X 0,Y 546.4,Z 349.755,A -85,B 0,C 180,E1 -3605.814,E2 -3605.814} C_VEL
LIN {X 0,Y 546.419,Z 318.024,A -85,B 0,C 180,E1 -3606.244,E2 -3606.244} C_VEL
LIN {X 0,Y 545.101,Z 313.588,A -85,B 0,C 180,E1 -3606.36,E2 -3606.36} C_VEL
LIN {X 0,Y 545.071,Z 313.592,A -85,B 0,C 180,E1 -3608.901,E2 -3608.901} C_VEL
LIN {X 0,Y 545.057,Z 313.589,A -85,B 0,C 180,E1 -3611.906,E2 -3611.906} C_VEL
LIN {X 0,Y 545.081,Z 313.587,A -85,B 0,C 180,E1 -3614.944,E2 -3614.944} C_VEL
LIN {X 0,Y 545.045,Z 313.592,A -85,B 0,C 180,E1 -3618.027,E2 -3618.027} C_VEL
LIN {X 0,Y 545.004,Z 313.601,A -85,B 0,C 180,E1 -3620.376,E2 -3620.376} C_VEL
LIN {X 0,Y 545.012,Z 313.595,A -85,B 0,C 180,E1 -3622.759,E2 -3622.759} C_VEL
LIN {X 0,Y 545.024,Z 313.591,A -85,B 0,C 180,E1 -3625.492,E2 -3625.492} C_VEL
LIN {X 0,Y 545.036,Z 313.593,A -85,B 0,C 180,E1 -3628.496,E2 -3628.496} C_VEL
LIN {X 0,Y 545.044,Z 313.588,A -85,B 0,C 180,E1 -3631.05,E2 -3631.05} C_VEL
LIN {X 0,Y 545.058,Z 313.589,A -85,B 0,C 180,E1 -3633.673,E2 -3633.673} C_VEL
LIN {X 0,Y 545.008,Z 313.595,A -85,B 0,C 180,E1 -3636.383,E2 -3636.383} C_VEL
LIN {X 0,Y 545.075,Z 313.584,A -85,B 0,C 180,E1 -3639.319,E2 -3639.319} C_VEL
LIN {X 0,Y 545.041,Z 313.593,A -85,B 0,C 180,E1 -3642.107,E2 -3642.107} C_VEL
LIN {X 0,Y 545.025,Z 313.589,A -85,B 0,C 180,E1 -3644.828,E2 -3644.828} C_VEL
LIN {X 0,Y 545.041,Z 313.59,A -85,B 0,C 180,E1 -3647.306,E2 -3647.306} C_VEL
LIN {X 0,Y 545.063,Z 313.593,A -85,B 0,C 180,E1 -3649.857,E2 -3649.857} C_VEL
LIN {X 0,Y 545.031,Z 313.589,A -85,B 0,C 180,E1 -3652.695,E2 -3652.695} C_VEL
LIN {X 0,Y 545.073,Z 313.592,A -85,B 0,C 180,E1 -3655.609,E2 -3655.609} C_VEL
LIN {X 0,Y 545.062,Z 313.586,A -85,B 0,C 180,E1 -3658.321,E2 -3658.321} C_VEL
LIN {X 0,Y 545.073,Z 313.591,A -85,B 0,C 180,E1 -3661.256,E2 -3661.256} C_VEL
LIN {X 0,Y 545.104,Z 313.767,A -85,B 0,C 180,E1 -3662.62,E2 -3662.62} C_VEL
LIN {X 0,Y 547.083,Z 323.628,A -85,B 0,C 180,E1 -3663.917,E2 -3663.917} C_VEL
LIN {X 0,Y 546.735,Z 345.133,A -85,B 0,C 180,E1 -3666.516,E2 -3666.516} C_VEL
LIN {X 0,Y 546.301,Z 369.868,A -85,B 0,C 180,E1 -3669.478,E2 -3669.478} C_VEL
LIN {X 0,Y 545.932,Z 396.097,A -85,B 0,C 180,E1 -3672.539,E2 -3672.539} C_VEL
LIN {X 0,Y 545.609,Z 421.106,A -85,B 0,C 180,E1 -3675.429,E2 -3675.429} C_VEL
LIN {X 0,Y 546.593,Z 429.067,A -85,B 0,C 180,E1 -3675.559,E2 -3675.559} C_VEL
LIN {X 0,Y 546.207,Z 530.935,A -85,B 0,C 180,E1 -3676.916,E2 -3676.916} C_VEL
LIN {X 0,Y 546.055,Z 544.21,A -85,B 0,C 180,E1 -3677.243,E2 -3677.243} C_VEL
LIN {X 0,Y 545.863,Z 557.484,A -85,B 0,C 180,E1 -3677.735,E2 -3677.735} C_VEL
LIN {X 0,Y 545.653,Z 570.028,A -85,B 0,C 180,E1 -3678.38,E2 -3678.38} C_VEL
LIN {X 0,Y 545.476,Z 581.482,A -85,B 0,C 180,E1 -3679.139,E2 -3679.139} C_VEL
LIN {X 0,Y 545.259,Z 591.644,A -85,B 0,C 180,E1 -3679.979,E2 -3679.979} C_VEL
LIN {X 0,Y 545.079,Z 600.784,A -85,B 0,C 180,E1 -3680.912,E2 -3680.912} C_VEL
LIN {X 0,Y 544.917,Z 609.687,A -85,B 0,C 180,E1 -3682.03,E2 -3682.03} C_VEL
LIN {X 0,Y 544.785,Z 616.847,A -85,B 0,C 180,E1 -3683.146,E2 -3683.146} C_VEL
LIN {X 0,Y 544.741,Z 623.365,A -85,B 0,C 180,E1 -3684.447,E2 -3684.447} C_VEL
LIN {X 0,Y 544.66,Z 627.676,A -85,B 0,C 180,E1 -3685.56,E2 -3685.56} C_VEL
LIN {X 0,Y 544.669,Z 629.958,A -85,B 0,C 180,E1 -3686.301,E2 -3686.301} C_VEL
LIN {X 0,Y 544.65,Z 631.807,A -85,B 0,C 180,E1 -3687.041,E2 -3687.041} C_VEL
LIN {X 0,Y 544.546,Z 634.183,A -85,B 0,C 180,E1 -3688.521,E2 -3688.521} C_VEL
LIN {X 0,Y 544.541,Z 635,A -85,B 0,C 180,E1 -3690,E2 -3690} C_VEL
LIN {X 0,Y 544.546,Z 634.184,A -85,B 0,C 180,E1 -3691.479,E2 -3691.479} C_VEL
LIN {X 0,Y 544.65,Z 631.81,A -85,B 0,C 180,E1 -3692.959,E2 -3692.959} C_VEL
LIN {X 0,Y 544.684,Z 628.896,A -85,B 0,C 180,E1 -3694.069,E2 -3694.069} C_VEL
LIN {X 0,Y 544.654,Z 624.948,A -85,B 0,C 180,E1 -3695.182,E2 -3695.182} C_VEL
LIN {X 0,Y 544.73,Z 619.644,A -85,B 0,C 180,E1 -3696.339,E2 -3696.339} C_VEL
LIN {X 0,Y 544.837,Z 613.467,A -85,B 0,C 180,E1 -3697.411,E2 -3697.411} C_VEL
LIN {X 0,Y 545.007,Z 605.478,A -85,B 0,C 180,E1 -3698.528,E2 -3698.528} C_VEL
LIN {X 0,Y 545.152,Z 597.334,A -85,B 0,C 180,E1 -3699.461,E2 -3699.461} C_VEL
LIN {X 0,Y 545.376,Z 587.398,A -85,B 0,C 180,E1 -3700.394,E2 -3700.394} C_VEL
LIN {X 0,Y 545.57,Z 576.593,A -85,B 0,C 180,E1 -3701.208,E2 -3701.208} C_VEL
LIN {X 0,Y 545.747,Z 565.172,A -85,B 0,C 180,E1 -3701.891,E2 -3701.891} C_VEL
LIN {X 0,Y 545.919,Z 552.973,A -85,B 0,C 180,E1 -3702.453,E2 -3702.453} C_VEL
LIN {X 0,Y 546.169,Z 540.174,A -85,B 0,C 180,E1 -3702.872,E2 -3702.872} C_VEL
LIN {X 0,Y 546.242,Z 528.105,A -85,B 0,C 180,E1 -3703.13,E2 -3703.13} C_VEL
LIN {X 0,Y 546.472,Z 427.556,A -85,B 0,C 180,E1 -3704.463,E2 -3704.463} C_VEL
LIN {X 0,Y 545.603,Z 420.944,A -85,B 0,C 180,E1 -3704.59,E2 -3704.59} C_VEL
LIN {X 0,Y 545.921,Z 392.766,A -85,B 0,C 180,E1 -3707.797,E2 -3707.797} C_VEL
LIN {X 0,Y 546.236,Z 365.591,A -85,B 0,C 180,E1 -3710.918,E2 -3710.918} C_VEL
LIN {X 0,Y 546.552,Z 339.354,A -85,B 0,C 180,E1 -3713.981,E2 -3713.981} C_VEL
LIN {X 0,Y 546.672,Z 322.999,A -85,B 0,C 180,E1 -3715.919,E2 -3715.919} C_VEL
LIN {X 0,Y 545.924,Z 317.775,A -85,B 0,C 180,E1 -3716.574,E2 -3716.574} C_VEL
LIN {X 0,Y 545.039,Z 313.594,A -85,B 0,C 180,E1 -3717.126,E2 -3717.126} C_VEL
LIN {X 0,Y 545.061,Z 313.589,A -85,B 0,C 180,E1 -3719.339,E2 -3719.339} C_VEL
LIN {X 0,Y 545.058,Z 313.591,A -85,B 0,C 180,E1 -3721.915,E2 -3721.915} C_VEL
LIN {X 0,Y 545.061,Z 313.593,A -85,B 0,C 180,E1 -3724.565,E2 -3724.565} C_VEL
LIN {X 0,Y 545.033,Z 313.589,A -85,B 0,C 180,E1 -3727.304,E2 -3727.304} C_VEL
LIN {X 0,Y 545.061,Z 313.594,A -85,B 0,C 180,E1 -3730.143,E2 -3730.143} C_VEL
LIN {X 0,Y 545.025,Z 313.591,A -85,B 0,C 180,E1 -3733.112,E2 -3733.112} C_VEL
LIN {X 0,Y 545.048,Z 313.595,A -85,B 0,C 180,E1 -3736.227,E2 -3736.227} C_VEL
LIN {X 0,Y 545.022,Z 313.591,A -85,B 0,C 180,E1 -3738.88,E2 -3738.88} C_VEL
LIN {X 0,Y 545.047,Z 313.593,A -85,B 0,C 180,E1 -3741.762,E2 -3741.762} C_VEL
LIN {X 0,Y 545.024,Z 313.591,A -85,B 0,C 180,E1 -3744.53,E2 -3744.53} C_VEL
LIN {X 0,Y 545.063,Z 313.586,A -85,B 0,C 180,E1 -3747.211,E2 -3747.211} C_VEL
LIN {X 0,Y 545.065,Z 313.594,A -85,B 0,C 180,E1 -3749.81,E2 -3749.81} C_VEL
LIN {X 0,Y 545.022,Z 313.591,A -85,B 0,C 180,E1 -3752.842,E2 -3752.842} C_VEL
LIN {X 0,Y 545.014,Z 313.6,A -85,B 0,C 180,E1 -3755.629,E2 -3755.629} C_VEL
LIN {X 0,Y 545.046,Z 313.59,A -85,B 0,C 180,E1 -3758.186,E2 -3758.186} C_VEL
LIN {X 0,Y 545.03,Z 313.594,A -85,B 0,C 180,E1 -3761.193,E2 -3761.193} C_VEL
LIN {X 0,Y 545.037,Z 313.597,A -85,B 0,C 180,E1 -3763.52,E2 -3763.52} C_VEL
LIN {X 0,Y 545.072,Z 313.591,A -85,B 0,C 180,E1 -3765.819,E2 -3765.819} C_VEL
LIN {X 0,Y 545.093,Z 313.608,A -85,B 0,C 180,E1 -3767.748,E2 -3767.748} C_VEL
LIN {X 0,Y 546.501,Z 318.819,A -85,B 0,C 180,E1 -3767.857,E2 -3767.857} C_VEL
LIN {X 0,Y 546.161,Z 402.153,A -85,B 0,C 180,E1 -3768.988,E2 -3768.988} C_VEL
LIN {X 0,Y 546.018,Z 415.275,A -85,B 0,C 180,E1 -3769.314,E2 -3769.314} C_VEL
LIN {X 0,Y 545.885,Z 428.342,A -85,B 0,C 180,E1 -3769.803,E2 -3769.803} C_VEL
LIN {X 0,Y 545.734,Z 439.297,A -85,B 0,C 180,E1 -3770.362,E2 -3770.362} C_VEL
LIN {X 0,Y 545.57,Z 448.156,A -85,B 0,C 180,E1 -3770.92,E2 -3770.92} C_VEL
LIN {X 0,Y 545.352,Z 457.801,A -85,B 0,C 180,E1 -3771.664,E2 -3771.664} C_VEL
LIN {X 0,Y 545.188,Z 465.809,A -85,B 0,C 180,E1 -3772.407,E2 -3772.407} C_VEL
LIN {X 0,Y 545.048,Z 472.615,A -85,B 0,C 180,E1 -3773.151,E2 -3773.151} C_VEL
LIN {X 0,Y 544.888,Z 479.723,A -85,B 0,C 180,E1 -3774.077,E2 -3774.077} C_VEL
LIN {X 0,Y 544.881,Z 485.657,A -85,B 0,C 180,E1 -3775.005,E2 -3775.005} C_VEL
LIN {X 0,Y 544.746,Z 490.694,A -85,B 0,C 180,E1 -3775.931,E2 -3775.931} C_VEL
LIN {X 0,Y 544.682,Z 495.567,A -85,B 0,C 180,E1 -3777.041,E2 -3777.041} C_VEL
LIN {X 0,Y 544.664,Z 499.335,A -85,B 0,C 180,E1 -3778.151,E2 -3778.151} C_VEL
LIN {X 0,Y 544.546,Z 502.091,A -85,B 0,C 180,E1 -3779.26,E2 -3779.26} C_VEL
LIN {X 0,Y 544.542,Z 503.449,A -85,B 0,C 180,E1 -3780,E2 -3780} C_VEL
LIN {X 0,Y 544.543,Z 504.35,A -85,B 0,C 180,E1 -3780.739,E2 -3780.739} C_VEL
LIN {X 0,Y 544.569,Z 504.959,A -85,B 0,C 180,E1 -3782.219,E2 -3782.219} C_VEL
LIN {X 0,Y 544.645,Z 504.658,A -85,B 0,C 180,E1 -3782.958,E2 -3782.958} C_VEL
LIN {X 0,Y 544.599,Z 502.886,A -85,B 0,C 180,E1 -3784.44,E2 -3784.44} C_VEL
LIN {X 0,Y 544.616,Z 501.365,A -85,B 0,C 180,E1 -3785.182,E2 -3785.182} C_VEL
LIN {X 0,Y 544.695,Z 497.02,A -85,B 0,C 180,E1 -3786.668,E2 -3786.668} C_VEL
LIN {X 0,Y 544.745,Z 492.483,A -85,B 0,C 180,E1 -3787.785,E2 -3787.785} C_VEL
LIN {X 0,Y 544.787,Z 487.801,A -85,B 0,C 180,E1 -3788.718,E2 -3788.718} C_VEL
LIN {X 0,Y 544.851,Z 482.168,A -85,B 0,C 180,E1 -3789.653,E2 -3789.653} C_VEL
LIN {X 0,Y 545.021,Z 475.435,A -85,B 0,C 180,E1 -3790.588,E2 -3790.588} C_VEL
LIN {X 0,Y 545.107,Z 468.832,A -85,B 0,C 180,E1 -3791.367,E2 -3791.367} C_VEL
LIN {X 0,Y 545.272,Z 460.535,A -85,B 0,C 180,E1 -3792.184,E2 -3792.184} C_VEL
LIN {X 0,Y 545.481,Z 451.309,A -85,B 0,C 180,E1 -3792.935,E2 -3792.935} C_VEL
LIN {X 0,Y 545.611,Z 443.023,A -85,B 0,C 180,E1 -3793.501,E2 -3793.501} C_VEL
LIN {X 0,Y 545.796,Z 432.85,A -85,B 0,C 180,E1 -3794.066,E2 -3794.066} C_VEL
LIN {X 0,Y 546.004,Z 423.268,A -85,B 0,C 180,E1 -3794.489,E2 -3794.489} C_VEL
LIN {X 0,Y 546.061,Z 412.786,A -85,B 0,C 180,E1 -3794.844,E2 -3794.844} C_VEL
LIN {X 0,Y 546.173,Z 401.189,A -85,B 0,C 180,E1 -3795.122,E2 -3795.122} C_VEL
LIN {X 0,Y 546.467,Z 318.083,A -85,B 0,C 180,E1 -3796.243,E2 -3796.243} C_VEL
LIN {X 0,Y 545.093,Z 313.588,A -85,B 0,C 180,E1 -3796.357,E2 -3796.357} C_VEL
LIN {X 0,Y 545.118,Z 313.578,A -85,B 0,C 180,E1 -3799.585,E2 -3799.585} C_VEL
LIN {X 0,Y 545.037,Z 313.596,A -85,B 0,C 180,E1 -3802.757,E2 -3802.757} C_VEL
LIN {X 0,Y 545.116,Z 313.58,A -85,B 0,C 180,E1 -3805.198,E2 -3805.198} C_VEL
LIN {X 0,Y 544.413,Z 313.667,A -85,B 0,C 180,E1 -3805.815,E2 -3805.815} C_VEL
LIN {X 0,Y 541.538,Z 314.03,A -85,B 0,C 180,E1 -3806.816,E2 -3806.816} C_VEL
LIN {X 0,Y 539.133,Z 314.327,A -85,B 0,C 180,E1 -3807.623,E2 -3807.623} C_VEL
LIN {X 0,Y 538.108,Z 314.455,A -85,B 0,C 180,E1 -3808.245,E2 -3808.245} C_VEL
LIN {X 0,Y 538.027,Z 314.463,A -85,B 0,C 180,E1 -3808.456,E2 -3808.456} C_VEL
LIN {X 0,Y 538.009,Z 314.464,A -85,B 0,C 180,E1 -3811.501,E2 -3811.501} C_VEL
LIN {X 0,Y 538.011,Z 314.467,A -85,B 0,C 180,E1 -3814.173,E2 -3814.173} C_VEL
LIN {X 0,Y 538.003,Z 314.465,A -85,B 0,C 180,E1 -3817.169,E2 -3817.169} C_VEL
LIN {X 0,Y 538.021,Z 314.463,A -85,B 0,C 180,E1 -3819.797,E2 -3819.797} C_VEL
LIN {X 0,Y 538.018,Z 314.467,A -85,B 0,C 180,E1 -3822.786,E2 -3822.786} C_VEL
LIN {X 0,Y 538.006,Z 314.465,A -85,B 0,C 180,E1 -3825.138,E2 -3825.138} C_VEL
LIN {X 0,Y 538.029,Z 314.467,A -85,B 0,C 180,E1 -3828.226,E2 -3828.226} C_VEL
LIN {X 0,Y 538.014,Z 314.463,A -85,B 0,C 180,E1 -3831.169,E2 -3831.169} C_VEL
LIN {X 0,Y 538.024,Z 314.467,A -85,B 0,C 180,E1 -3834.084,E2 -3834.084} C_VEL
LIN {X 0,Y 538.03,Z 314.465,A -85,B 0,C 180,E1 -3836.727,E2 -3836.727} C_VEL
LIN {X 0,Y 538.024,Z 314.462,A -85,B 0,C 180,E1 -3839.556,E2 -3839.556} C_VEL
LIN {X 0,Y 538.042,Z 314.464,A -85,B 0,C 180,E1 -3841.95,E2 -3841.95} C_VEL
LIN {X 0,Y 538.07,Z 314.462,A -85,B 0,C 180,E1 -3844.467,E2 -3844.467} C_VEL
LIN {X 0,Y 538.021,Z 314.463,A -85,B 0,C 180,E1 -3846.928,E2 -3846.928} C_VEL
LIN {X 0,Y 538.077,Z 314.463,A -85,B 0,C 180,E1 -3850.148,E2 -3850.148} C_VEL
LIN {X 0,Y 538.022,Z 314.462,A -85,B 0,C 180,E1 -3853.299,E2 -3853.299} C_VEL
LIN {X 0,Y 538.062,Z 314.459,A -85,B 0,C 180,E1 -3855.631,E2 -3855.631} C_VEL
LIN {X 0,Y 538.075,Z 314.457,A -85,B 0,C 180,E1 -3858.702,E2 -3858.702} C_VEL
LIN {X 0,Y 538.083,Z 314.458,A -85,B 0,C 180,E1 -3861.74,E2 -3861.74} C_VEL
LIN {X 0,Y 538.159,Z 314.446,A -85,B 0,C 180,E1 -3864.755,E2 -3864.755} C_VEL
LIN {X 0,Y 538.168,Z 314.449,A -85,B 0,C 180,E1 -3867.755,E2 -3867.755} C_VEL
LIN {X 0,Y 538.181,Z 314.443,A -85,B 0,C 180,E1 -3870.748,E2 -3870.748} C_VEL
LIN {X 0,Y 538.136,Z 314.448,A -85,B 0,C 180,E1 -3872.995,E2 -3872.995} C_VEL
LIN {X 0,Y 538.122,Z 314.458,A -85,B 0,C 180,E1 -3875.997,E2 -3875.997} C_VEL
LIN {X 0,Y 538.066,Z 314.457,A -85,B 0,C 180,E1 -3879.018,E2 -3879.018} C_VEL
LIN {X 0,Y 538.082,Z 314.462,A -85,B 0,C 180,E1 -3882.063,E2 -3882.063} C_VEL
LIN {X 0,Y 538.044,Z 314.46,A -85,B 0,C 180,E1 -3885.144,E2 -3885.144} C_VEL
LIN {X 0,Y 538.032,Z 314.464,A -85,B 0,C 180,E1 -3888.27,E2 -3888.27} C_VEL
LIN {X 0,Y 538.038,Z 314.46,A -85,B 0,C 180,E1 -3890.652,E2 -3890.652} C_VEL
LIN {X 0,Y 538.023,Z 314.47,A -85,B 0,C 180,E1 -3893.888,E2 -3893.888} C_VEL
LIN {X 0,Y 538.041,Z 314.461,A -85,B 0,C 180,E1 -3896.367,E2 -3896.367} C_VEL
LIN {X 0,Y 538.03,Z 314.462,A -85,B 0,C 180,E1 -3898.934,E2 -3898.934} C_VEL
LIN {X 0,Y 538.014,Z 314.47,A -85,B 0,C 180,E1 -3901.889,E2 -3901.889} C_VEL
LIN {X 0,Y 538.03,Z 314.461,A -85,B 0,C 180,E1 -3904.621,E2 -3904.621} C_VEL
LIN {X 0,Y 538.006,Z 314.467,A -85,B 0,C 180,E1 -3907.171,E2 -3907.171} C_VEL
LIN {X 0,Y 538.026,Z 314.469,A -85,B 0,C 180,E1 -3909.797,E2 -3909.797} C_VEL
LIN {X 0,Y 538.019,Z 314.463,A -85,B 0,C 180,E1 -3912.787,E2 -3912.787} C_VEL
LIN {X 0,Y 538.03,Z 314.465,A -85,B 0,C 180,E1 -3915.926,E2 -3915.926} C_VEL
LIN {X 0,Y 538.049,Z 314.464,A -85,B 0,C 180,E1 -3919.253,E2 -3919.253} C_VEL
LIN {X 0,Y 537.993,Z 314.467,A -85,B 0,C 180,E1 -3922.123,E2 -3922.123} C_VEL
LIN {X 0,Y 537.999,Z 314.467,A -85,B 0,C 180,E1 -3924.916,E2 -3924.916} C_VEL
LIN {X 0,Y 538.019,Z 314.47,A -85,B 0,C 180,E1 -3927.618,E2 -3927.618} C_VEL
LIN {X 0,Y 538.017,Z 314.463,A -85,B 0,C 180,E1 -3930.239,E2 -3930.239} C_VEL
LIN {X 0,Y 538.054,Z 314.46,A -85,B 0,C 180,E1 -3932.796,E2 -3932.796} C_VEL
LIN {X 0,Y 538.046,Z 314.467,A -85,B 0,C 180,E1 -3935.293,E2 -3935.293} C_VEL
LIN {X 0,Y 538.026,Z 314.47,A -85,B 0,C 180,E1 -3937.556,E2 -3937.556} C_VEL
LIN {X 0,Y 539.521,Z 319.322,A -85,B 0,C 180,E1 -3937.68,E2 -3937.68} C_VEL
LIN {X 0,Y 539.276,Z 402.228,A -85,B 0,C 180,E1 -3938.824,E2 -3938.824} C_VEL
LIN {X 0,Y 539.17,Z 414.522,A -85,B 0,C 180,E1 -3939.12,E2 -3939.12} C_VEL
LIN {X 0,Y 539.001,Z 426.862,A -85,B 0,C 180,E1 -3939.563,E2 -3939.563} C_VEL
LIN {X 0,Y 538.799,Z 439.186,A -85,B 0,C 180,E1 -3940.176,E2 -3940.176} C_VEL
LIN {X 0,Y 538.584,Z 449.845,A -85,B 0,C 180,E1 -3940.862,E2 -3940.862} C_VEL
LIN {X 0,Y 538.376,Z 458.554,A -85,B 0,C 180,E1 -3941.545,E2 -3941.545} C_VEL
LIN {X 0,Y 538.239,Z 466.331,A -85,B 0,C 180,E1 -3942.274,E2 -3942.274} C_VEL
LIN {X 0,Y 538.061,Z 473.825,A -85,B 0,C 180,E1 -3943.105,E2 -3943.105} C_VEL
LIN {X 0,Y 537.915,Z 481.108,A -85,B 0,C 180,E1 -3944.076,E2 -3944.076} C_VEL
LIN {X 0,Y 537.761,Z 487.623,A -85,B 0,C 180,E1 -3945.131,E2 -3945.131} C_VEL
LIN {X 0,Y 537.708,Z 492.066,A -85,B 0,C 180,E1 -3946.008,E2 -3946.008} C_VEL
LIN {X 0,Y 537.587,Z 496.822,A -85,B 0,C 180,E1 -3947.159,E2 -3947.159} C_VEL
LIN {X 0,Y 537.566,Z 500.429,A -85,B 0,C 180,E1 -3948.309,E2 -3948.309} C_VEL
LIN {X 0,Y 537.498,Z 503.003,A -85,B 0,C 180,E1 -3949.453,E2 -3949.453} C_VEL
LIN {X 0,Y 537.498,Z 504.997,A -85,B 0,C 180,E1 -3950.973,E2 -3950.973} C_VEL
LIN {X 0,Y 537.54,Z 505.261,A -85,B 0,C 180,E1 -3952.488,E2 -3952.488} C_VEL
LIN {X 0,Y 537.574,Z 504.602,A -85,B 0,C 180,E1 -3953.513,E2 -3953.513} C_VEL
LIN {X 0,Y 537.525,Z 502.811,A -85,B 0,C 180,E1 -3954.749,E2 -3954.749} C_VEL
LIN {X 0,Y 537.603,Z 500.2,A -85,B 0,C 180,E1 -3955.877,E2 -3955.877} C_VEL
LIN {X 0,Y 537.629,Z 496.613,A -85,B 0,C 180,E1 -3957.003,E2 -3957.003} C_VEL
LIN {X 0,Y 537.683,Z 491.945,A -85,B 0,C 180,E1 -3958.128,E2 -3958.128} C_VEL
LIN {X 0,Y 537.799,Z 487.116,A -85,B 0,C 180,E1 -3959.064,E2 -3959.064} C_VEL
LIN {X 0,Y 537.93,Z 481.316,A -85,B 0,C 180,E1 -3960,E2 -3960} C_VEL
LIN {X 0,Y 538.056,Z 474.367,A -85,B 0,C 180,E1 -3960.936,E2 -3960.936} C_VEL
LIN {X 0,Y 538.241,Z 465.981,A -85,B 0,C 180,E1 -3961.871,E2 -3961.871} C_VEL
LIN {X 0,Y 538.499,Z 455.679,A -85,B 0,C 180,E1 -3962.806,E2 -3962.806} C_VEL
LIN {X 0,Y 538.745,Z 443.822,A -85,B 0,C 180,E1 -3963.647,E2 -3963.647} C_VEL
LIN {X 0,Y 538.928,Z 433.836,A -85,B 0,C 180,E1 -3964.207,E2 -3964.207} C_VEL
LIN {X 0,Y 539.027,Z 423.271,A -85,B 0,C 180,E1 -3964.675,E2 -3964.675} C_VEL
LIN {X 0,Y 539.155,Z 411.852,A -85,B 0,C 180,E1 -3965.048,E2 -3965.048} C_VEL
LIN {X 0,Y 539.246,Z 400.056,A -85,B 0,C 180,E1 -3965.305,E2 -3965.305} C_VEL
LIN {X 0,Y 539.535,Z 319.345,A -85,B 0,C 180,E1 -3966.412,E2 -3966.412} C_VEL
LIN {X 0,Y 538.04,Z 314.468,A -85,B 0,C 180,E1 -3966.536,E2 -3966.536} C_VEL
LIN {X 0,Y 538.028,Z 314.468,A -85,B 0,C 180,E1 -3969.019,E2 -3969.019} C_VEL
LIN {X 0,Y 538.013,Z 314.467,A -85,B 0,C 180,E1 -3972.064,E2 -3972.064} C_VEL
LIN {X 0,Y 538.042,Z 314.462,A -85,B 0,C 180,E1 -3975.144,E2 -3975.144} C_VEL
LIN {X 0,Y 537.995,Z 314.474,A -85,B 0,C 180,E1 -3978.272,E2 -3978.272} C_VEL
LIN {X 0,Y 537.972,Z 314.475,A -85,B 0,C 180,E1 -3980.654,E2 -3980.654} C_VEL
LIN {X 0,Y 538,Z 314.466,A -85,B 0,C 180,E1 -3983.073,E2 -3983.073} C_VEL
LIN {X 0,Y 537.985,Z 314.469,A -85,B 0,C 180,E1 -3985.658,E2 -3985.658} C_VEL
LIN {X 0,Y 537.974,Z 314.475,A -85,B 0,C 180,E1 -3988.054,E2 -3988.054} C_VEL
LIN {X 0,Y 538,Z 314.468,A -85,B 0,C 180,E1 -3990.629,E2 -3990.629} C_VEL
LIN {X 0,Y 538.025,Z 314.462,A -85,B 0,C 180,E1 -3993.278,E2 -3993.278} C_VEL
LIN {X 0,Y 537.961,Z 314.477,A -85,B 0,C 180,E1 -3996.008,E2 -3996.008} C_VEL
LIN {X 0,Y 538.012,Z 314.462,A -85,B 0,C 180,E1 -3998.831,E2 -3998.831} C_VEL
LIN {X 0,Y 537.99,Z 314.473,A -85,B 0,C 180,E1 -4001.873,E2 -4001.873} C_VEL
LIN {X 0,Y 537.998,Z 314.465,A -85,B 0,C 180,E1 -4004.864,E2 -4004.864} C_VEL
LIN {X 0,Y 537.991,Z 314.468,A -85,B 0,C 180,E1 -4007.211,E2 -4007.211} C_VEL
LIN {X 0,Y 538.015,Z 314.464,A -85,B 0,C 180,E1 -4010.418,E2 -4010.418} C_VEL
LIN {X 0,Y 537.996,Z 314.467,A -85,B 0,C 180,E1 -4013.064,E2 -4013.064} C_VEL
LIN {X 0,Y 538.016,Z 314.469,A -85,B 0,C 180,E1 -4015.826,E2 -4015.826} C_VEL
LIN {X 0,Y 538.013,Z 314.464,A -85,B 0,C 180,E1 -4018.499,E2 -4018.499} C_VEL
LIN {X 0,Y 538.022,Z 314.468,A -85,B 0,C 180,E1 -4021.097,E2 -4021.097} C_VEL
LIN {X 0,Y 538.062,Z 314.537,A -85,B 0,C 180,E1 -4022.404,E2 -4022.404} C_VEL
LIN {X 0,Y 540.203,Z 325.392,A -85,B 0,C 180,E1 -4023.856,E2 -4023.856} C_VEL
LIN {X 0,Y 539.735,Z 349.492,A -85,B 0,C 180,E1 -4026.803,E2 -4026.803} C_VEL
LIN {X 0,Y 539.264,Z 374.869,A -85,B 0,C 180,E1 -4029.881,E2 -4029.881} C_VEL
LIN {X 0,Y 538.877,Z 399.112,A -85,B 0,C 180,E1 -4032.74,E2 -4032.74} C_VEL
LIN {X 0,Y 538.559,Z 420.532,A -85,B 0,C 180,E1 -4035.246,E2 -4035.246} C_VEL
LIN {X 0,Y 539.681,Z 430.048,A -85,B 0,C 180,E1 -4035.403,E2 -4035.403} C_VEL
LIN {X 0,Y 539.292,Z 529.873,A -85,B 0,C 180,E1 -4036.745,E2 -4036.745} C_VEL
LIN {X 0,Y 539.124,Z 542.704,A -85,B 0,C 180,E1 -4037.052,E2 -4037.052} C_VEL
LIN {X 0,Y 538.918,Z 555.842,A -85,B 0,C 180,E1 -4037.526,E2 -4037.526} C_VEL
LIN {X 0,Y 538.704,Z 567.349,A -85,B 0,C 180,E1 -4038.087,E2 -4038.087} C_VEL
LIN {X 0,Y 538.531,Z 578.784,A -85,B 0,C 180,E1 -4038.806,E2 -4038.806} C_VEL
LIN {X 0,Y 538.272,Z 589.523,A -85,B 0,C 180,E1 -4039.658,E2 -4039.658} C_VEL
LIN {X 0,Y 538.067,Z 599.111,A -85,B 0,C 180,E1 -4040.603,E2 -4040.603} C_VEL
LIN {X 0,Y 537.921,Z 606.959,A -85,B 0,C 180,E1 -4041.548,E2 -4041.548} C_VEL
LIN {X 0,Y 537.755,Z 614.62,A -85,B 0,C 180,E1 -4042.679,E2 -4042.679} C_VEL
LIN {X 0,Y 537.693,Z 621.679,A -85,B 0,C 180,E1 -4043.998,E2 -4043.998} C_VEL
LIN {X 0,Y 537.541,Z 626.372,A -85,B 0,C 180,E1 -4045.125,E2 -4045.125} C_VEL
LIN {X 0,Y 537.591,Z 629.957,A -85,B 0,C 180,E1 -4046.252,E2 -4046.252} C_VEL
LIN {X 0,Y 537.551,Z 631.806,A -85,B 0,C 180,E1 -4047.002,E2 -4047.002} C_VEL
LIN {X 0,Y 537.451,Z 634.182,A -85,B 0,C 180,E1 -4048.501,E2 -4048.501} C_VEL
LIN {X 0,Y 537.442,Z 635,A -85,B 0,C 180,E1 -4050,E2 -4050} C_VEL
LIN {X 0,Y 537.451,Z 634.184,A -85,B 0,C 180,E1 -4051.499,E2 -4051.499} C_VEL
LIN {X 0,Y 537.551,Z 631.81,A -85,B 0,C 180,E1 -4052.998,E2 -4052.998} C_VEL
LIN {X 0,Y 537.603,Z 628.895,A -85,B 0,C 180,E1 -4054.123,E2 -4054.123} C_VEL
LIN {X 0,Y 537.588,Z 624.948,A -85,B 0,C 180,E1 -4055.251,E2 -4055.251} C_VEL
LIN {X 0,Y 537.645,Z 620.126,A -85,B 0,C 180,E1 -4056.326,E2 -4056.326} C_VEL
LIN {X 0,Y 537.791,Z 613.467,A -85,B 0,C 180,E1 -4057.509,E2 -4057.509} C_VEL
LIN {X 0,Y 537.973,Z 605.477,A -85,B 0,C 180,E1 -4058.64,E2 -4058.64} C_VEL
LIN {X 0,Y 538.143,Z 597.333,A -85,B 0,C 180,E1 -4059.585,E2 -4059.585} C_VEL
LIN {X 0,Y 538.384,Z 587.379,A -85,B 0,C 180,E1 -4060.53,E2 -4060.53} C_VEL
LIN {X 0,Y 538.566,Z 577.454,A -85,B 0,C 180,E1 -4061.288,E2 -4061.288} C_VEL
LIN {X 0,Y 538.727,Z 566.466,A -85,B 0,C 180,E1 -4061.957,E2 -4061.957} C_VEL
LIN {X 0,Y 538.946,Z 553.444,A -85,B 0,C 180,E1 -4062.569,E2 -4062.569} C_VEL
LIN {X 0,Y 539.16,Z 540.952,A -85,B 0,C 180,E1 -4062.994,E2 -4062.994} C_VEL
LIN {X 0,Y 539.295,Z 528.062,A -85,B 0,C 180,E1 -4063.279,E2 -4063.279} C_VEL
LIN {X 0,Y 539.492,Z 427.7,A -85,B 0,C 180,E1 -4064.625,E2 -4064.625} C_VEL
LIN {X 0,Y 538.537,Z 420.064,A -85,B 0,C 180,E1 -4064.764,E2 -4064.764} C_VEL
LIN {X 0,Y 538.897,Z 391.086,A -85,B 0,C 180,E1 -4068.105,E2 -4068.105} C_VEL
LIN {X 0,Y 539.252,Z 364.522,A -85,B 0,C 180,E1 -4071.202,E2 -4071.202} C_VEL
LIN {X 0,Y 539.564,Z 340.575,A -85,B 0,C 180,E1 -4074.037,E2 -4074.037} C_VEL
LIN {X 0,Y 539.732,Z 323.95,A -85,B 0,C 180,E1 -4076.042,E2 -4076.042} C_VEL
LIN {X 0,Y 538.02,Z 314.468,A -85,B 0,C 180,E1 -4077.287,E2 -4077.287} C_VEL
LIN {X 0,Y 538.016,Z 314.467,A -85,B 0,C 180,E1 -4079.761,E2 -4079.761} C_VEL
LIN {X 0,Y 538.02,Z 314.472,A -85,B 0,C 180,E1 -4082.383,E2 -4082.383} C_VEL
LIN {X 0,Y 537.996,Z 314.467,A -85,B 0,C 180,E1 -4085.085,E2 -4085.085} C_VEL
LIN {X 0,Y 537.991,Z 314.47,A -85,B 0,C 180,E1 -4087.878,E2 -4087.878} C_VEL
LIN {X 0,Y 538.003,Z 314.468,A -85,B 0,C 180,E1 -4090.78,E2 -4090.78} C_VEL
LIN {X 0,Y 538.013,Z 314.471,A -85,B 0,C 180,E1 -4094.072,E2 -4094.072} C_VEL
LIN {X 0,Y 537.982,Z 314.467,A -85,B 0,C 180,E1 -4097.018,E2 -4097.018} C_VEL
LIN {X 0,Y 538.004,Z 314.465,A -85,B 0,C 180,E1 -4099.259,E2 -4099.259} C_VEL
LIN {X 0,Y 537.983,Z 314.474,A -85,B 0,C 180,E1 -4102.121,E2 -4102.121} C_VEL
LIN {X 0,Y 537.997,Z 314.467,A -85,B 0,C 180,E1 -4105.385,E2 -4105.385} C_VEL
LIN {X 0,Y 538.001,Z 314.471,A -85,B 0,C 180,E1 -4108.115,E2 -4108.115} C_VEL
LIN {X 0,Y 537.987,Z 314.468,A -85,B 0,C 180,E1 -4111.095,E2 -4111.095} C_VEL
LIN {X 0,Y 537.977,Z 314.476,A -85,B 0,C 180,E1 -4113.63,E2 -4113.63} C_VEL
LIN {X 0,Y 538.009,Z 314.468,A -85,B 0,C 180,E1 -4116.122,E2 -4116.122} C_VEL
LIN {X 0,Y 537.988,Z 314.468,A -85,B 0,C 180,E1 -4118.544,E2 -4118.544} C_VEL
LIN {X 0,Y 537.987,Z 314.469,A -85,B 0,C 180,E1 -4120.938,E2 -4120.938} C_VEL
LIN {X 0,Y 537.986,Z 314.474,A -85,B 0,C 180,E1 -4123.297,E2 -4123.297} C_VEL
LIN {X 0,Y 538.045,Z 314.469,A -85,B 0,C 180,E1 -4125.63,E2 -4125.63} C_VEL
LIN {X 0,Y 538.027,Z 314.47,A -85,B 0,C 180,E1 -4127.565,E2 -4127.565} C_VEL
LIN {X 0,Y 539.649,Z 320.226,A -85,B 0,C 180,E1 -4127.692,E2 -4127.692} C_VEL
LIN {X 0,Y 539.209,Z 403.338,A -85,B 0,C 180,E1 -4128.844,E2 -4128.844} C_VEL
LIN {X 0,Y 539.102,Z 416.383,A -85,B 0,C 180,E1 -4129.175,E2 -4129.175} C_VEL
LIN {X 0,Y 538.974,Z 429.408,A -85,B 0,C 180,E1 -4129.671,E2 -4129.671} C_VEL
LIN {X 0,Y 538.803,Z 440.355,A -85,B 0,C 180,E1 -4130.237,E2 -4130.237} C_VEL
LIN {X 0,Y 538.596,Z 450.485,A -85,B 0,C 180,E1 -4130.896,E2 -4130.896} C_VEL
LIN {X 0,Y 538.415,Z 459.903,A -85,B 0,C 180,E1 -4131.65,E2 -4131.65} C_VEL
LIN {X 0,Y 538.202,Z 468.635,A -85,B 0,C 180,E1 -4132.496,E2 -4132.496} C_VEL
LIN {X 0,Y 538.057,Z 477.164,A -85,B 0,C 180,E1 -4133.503,E2 -4133.503} C_VEL
LIN {X 0,Y 537.861,Z 485.586,A -85,B 0,C 180,E1 -4134.752,E2 -4134.752} C_VEL
LIN {X 0,Y 537.744,Z 491.562,A -85,B 0,C 180,E1 -4135.878,E2 -4135.878} C_VEL
LIN {X 0,Y 537.632,Z 496.313,A -85,B 0,C 180,E1 -4137.002,E2 -4137.002} C_VEL
LIN {X 0,Y 537.615,Z 499.969,A -85,B 0,C 180,E1 -4138.127,E2 -4138.127} C_VEL
LIN {X 0,Y 537.47,Z 502.651,A -85,B 0,C 180,E1 -4139.25,E2 -4139.25} C_VEL
LIN {X 0,Y 537.46,Z 503.954,A -85,B 0,C 180,E1 -4140,E2 -4140} C_VEL
LIN {X 0,Y 537.458,Z 504.827,A -85,B 0,C 180,E1 -4140.749,E2 -4140.749} C_VEL
LIN {X 0,Y 537.487,Z 505.365,A -85,B 0,C 180,E1 -4142.248,E2 -4142.248} C_VEL
LIN {X 0,Y 537.574,Z 505.062,A -85,B 0,C 180,E1 -4142.997,E2 -4142.997} C_VEL
LIN {X 0,Y 537.528,Z 503.275,A -85,B 0,C 180,E1 -4144.499,E2 -4144.499} C_VEL
LIN {X 0,Y 537.54,Z 501.794,A -85,B 0,C 180,E1 -4145.251,E2 -4145.251} C_VEL
LIN {X 0,Y 537.646,Z 497.464,A -85,B 0,C 180,E1 -4146.756,E2 -4146.756} C_VEL
LIN {X 0,Y 537.699,Z 492.976,A -85,B 0,C 180,E1 -4147.888,E2 -4147.888} C_VEL
LIN {X 0,Y 537.811,Z 487.26,A -85,B 0,C 180,E1 -4149.022,E2 -4149.022} C_VEL
LIN {X 0,Y 537.895,Z 481.416,A -85,B 0,C 180,E1 -4149.969,E2 -4149.969} C_VEL
LIN {X 0,Y 538.055,Z 474.366,A -85,B 0,C 180,E1 -4150.917,E2 -4150.917} C_VEL
LIN {X 0,Y 538.205,Z 467.275,A -85,B 0,C 180,E1 -4151.717,E2 -4151.717} C_VEL
LIN {X 0,Y 538.375,Z 458.651,A -85,B 0,C 180,E1 -4152.534,E2 -4152.534} C_VEL
LIN {X 0,Y 538.583,Z 448.882,A -85,B 0,C 180,E1 -4153.296,E2 -4153.296} C_VEL
LIN {X 0,Y 538.855,Z 436.556,A -85,B 0,C 180,E1 -4154.058,E2 -4154.058} C_VEL
LIN {X 0,Y 539.087,Z 424.131,A -85,B 0,C 180,E1 -4154.63,E2 -4154.63} C_VEL
LIN {X 0,Y 539.161,Z 412.834,A -85,B 0,C 180,E1 -4155.015,E2 -4155.015} C_VEL
LIN {X 0,Y 539.271,Z 400.449,A -85,B 0,C 180,E1 -4155.3,E2 -4155.3} C_VEL
LIN {X 0,Y 539.462,Z 319.144,A -85,B 0,C 180,E1 -4156.417,E2 -4156.417} C_VEL
LIN {X 0,Y 538.034,Z 314.469,A -85,B 0,C 180,E1 -4156.529,E2 -4156.529} C_VEL
LIN {X 0,Y 538.086,Z 314.455,A -85,B 0,C 180,E1 -4159.881,E2 -4159.881} C_VEL
LIN {X 0,Y 538.014,Z 314.466,A -85,B 0,C 180,E1 -4163.071,E2 -4163.071} C_VEL
LIN {X 0,Y 538.044,Z 314.459,A -85,B 0,C 180,E1 -4165.672,E2 -4165.672} C_VEL
LIN {X 0,Y 538.027,Z 314.463,A -85,B 0,C 180,E1 -4168.456,E2 -4168.456} C_VEL
LIN {X 0,Y 537.358,Z 314.549,A -85,B 0,C 180,E1 -4169.081,E2 -4169.081} C_VEL
LIN {X 0,Y 534.474,Z 314.906,A -85,B 0,C 180,E1 -4170.096,E2 -4170.096} C_VEL
LIN {X 0,Y 532.047,Z 315.211,A -85,B 0,C 180,E1 -4170.912,E2 -4170.912} C_VEL
LIN {X 0,Y 531.024,Z 315.334,A -85,B 0,C 180,E1 -4171.544,E2 -4171.544} C_VEL
LIN {X 0,Y 530.952,Z 315.343,A -85,B 0,C 180,E1 -4171.757,E2 -4171.757} C_VEL
LIN {X 0,Y 530.968,Z 315.345,A -85,B 0,C 180,E1 -4174.85,E2 -4174.85} C_VEL
LIN {X 0,Y 530.965,Z 315.341,A -85,B 0,C 180,E1 -4177.507,E2 -4177.507} C_VEL
LIN {X 0,Y 530.98,Z 315.347,A -85,B 0,C 180,E1 -4180.433,E2 -4180.433} C_VEL
LIN {X 0,Y 530.963,Z 315.341,A -85,B 0,C 180,E1 -4183.494,E2 -4183.494} C_VEL
LIN {X 0,Y 530.953,Z 315.351,A -85,B 0,C 180,E1 -4186.504,E2 -4186.504} C_VEL
LIN {X 0,Y 530.982,Z 315.341,A -85,B 0,C 180,E1 -4188.976,E2 -4188.976} C_VEL
LIN {X 0,Y 530.957,Z 315.342,A -85,B 0,C 180,E1 -4191.529,E2 -4191.529} C_VEL
LIN {X 0,Y 530.977,Z 315.348,A -85,B 0,C 180,E1 -4194.382,E2 -4194.382} C_VEL
LIN {X 0,Y 530.969,Z 315.341,A -85,B 0,C 180,E1 -4197.133,E2 -4197.133} C_VEL
LIN {X 0,Y 530.968,Z 315.343,A -85,B 0,C 180,E1 -4199.803,E2 -4199.803} C_VEL
LIN {X 0,Y 531.013,Z 315.342,A -85,B 0,C 180,E1 -4202.467,E2 -4202.467} C_VEL
LIN {X 0,Y 531.004,Z 315.337,A -85,B 0,C 180,E1 -4204.942,E2 -4204.942} C_VEL
LIN {X 0,Y 530.969,Z 315.349,A -85,B 0,C 180,E1 -4208.247,E2 -4208.247} C_VEL
LIN {X 0,Y 530.994,Z 315.34,A -85,B 0,C 180,E1 -4210.677,E2 -4210.677} C_VEL
LIN {X 0,Y 530.983,Z 315.339,A -85,B 0,C 180,E1 -4213.071,E2 -4213.071} C_VEL
LIN {X 0,Y 531.017,Z 315.335,A -85,B 0,C 180,E1 -4215.436,E2 -4215.436} C_VEL
LIN {X 0,Y 531.035,Z 315.336,A -85,B 0,C 180,E1 -4218.55,E2 -4218.55} C_VEL
LIN {X 0,Y 531.053,Z 315.333,A -85,B 0,C 180,E1 -4221.63,E2 -4221.63} C_VEL
LIN {X 0,Y 531.119,Z 315.324,A -85,B 0,C 180,E1 -4224.685,E2 -4224.685} C_VEL
LIN {X 0,Y 531.139,Z 315.324,A -85,B 0,C 180,E1 -4227.725,E2 -4227.725} C_VEL
LIN {X 0,Y 531.151,Z 315.319,A -85,B 0,C 180,E1 -4230.758,E2 -4230.758} C_VEL
LIN {X 0,Y 531.103,Z 315.324,A -85,B 0,C 180,E1 -4233.034,E2 -4233.034} C_VEL
LIN {X 0,Y 531.082,Z 315.334,A -85,B 0,C 180,E1 -4236.077,E2 -4236.077} C_VEL
LIN {X 0,Y 531.027,Z 315.334,A -85,B 0,C 180,E1 -4239.138,E2 -4239.138} C_VEL
